// TwinCAT 3 PLC project RobustSolutionDemoProject
// ProgramVersion: 3.1.4026.24
// libraries:
//   [RobustSolution], * (BATW)
//   Tc2_MC2, * (Beckhoff Automation GmbH)
//   Tc2_Standard, * (Beckhoff Automation GmbH)
//   Tc2_System, * (Beckhoff Automation GmbH)
// project tree:
//   GVLs/ GVL_IO.TcGVL (not stored), GVL_Module.TcGVL (not stored), GVL_ShareMemory.TcGVL
//   / PlcTask.TcTTO
//   POUs/10_Chamber1/DUTs/Ctrl Status Interface/ ST_Chamber1_CtrlStatus.TcDUT (not stored), ST_Chamber1_ServiceCtrl.TcDUT, ST_Chamber1_ServiceParam.TcDUT, ST_Chamber1_ServiceStatus.TcDUT
//   POUs/10_Chamber1/DUTs/External IO/ ST_Chamber1_Signal_In.TcDUT, ST_Chamber1_Signal_Out.TcDUT
//   POUs/10_Chamber1/DUTs/ E_Chamber1ErrorCode.TcDUT, E_Chamber1ServiceId.TcDUT
//   POUs/10_Chamber1/DUTs/Service Param/Door/ ST_Chamber1DoorCloseParam.TcDUT, ST_Chamber1DoorOpenParam.TcDUT
//   POUs/10_Chamber1/DUTs/Service Param/Endpoint1PrepareWaferTransfer/ E_Ch1Ep1PrepareWaferTransferStep.TcDUT, ST_ChEp1PrepareWaferTransferParam.TcDUT
//   POUs/10_Chamber1/DUTs/Service Param/LiftAxis/ ST_Chamber1LiftPinAxisMoveAbsParam.TcDUT (not stored), ST_Chamber1LiftPinAxisMoveVelParam.TcDUT (not stored)
//   POUs/10_Chamber1/DUTs/Service Param/PreparePosition/ E_Chamber1PreparePositionStep.TcDUT, ST_Chamber1PreparePositionParam.TcDUT
//   POUs/10_Chamber1/DUTs/Service Param/SpinAxis/ ST_Chamber1SpinAxisJogParam.TcDUT (not stored), ST_Chamber1SpinAxisMoveAbsParam.TcDUT (not stored), ST_Chamber1SpinAxisMoveVelParam.TcDUT (not stored)
//   POUs/10_Chamber1/DUTs/Service Param/Vacuum/ ST_Chamber1VacuumOffParam.TcDUT, ST_Chamber1VacuumOnParam.TcDUT
//   POUs/10_Chamber1/ FB_Chamber1ModuleConfigurationAdapter.TcPOU, FB_Chamber1_Module.TcPOU
//   POUs/10_Chamber1/Services/Door/ FB_Chamber1Endpoint1DoorCloseService.TcPOU, FB_Chamber1Endpoint1DoorOpenService.TcPOU
//   POUs/10_Chamber1/Services/ FB_Chamber1PreparePositionService.TcPOU, FB_Chamber1Ep1PrepareWaferTransfer.TcPOU
//   POUs/10_Chamber1/Services/LiftAxis/ FB_Chamber1LiftPinAxisMoveAbsServices.TcPOU, FB_Chamber1LiftPinAxisMoveVelCCWServices.TcPOU, FB_Chamber1LiftPinAxisMoveVelCWServices.TcPOU
//   POUs/10_Chamber1/Services/SpinAxis/ FB_Chamber1SpinAxisJogCWServices.TcPOU, FB_Chamber1SpinAxisMoveAbsServices.TcPOU, FB_Chamber1SpinAxisMoveVelCWServices.TcPOU
//   POUs/10_Chamber1/Services/Vacuum/ FB_Chamber1VacuumOnService.TcPOU, FB_Chamber1VacuumOffService.TcPOU
//   POUs/ FB_ConfigRoot.TcPOU, MAIN.TcPOU (not stored)
// (motion and I/O tree: see PLC project robustsolutionframework)
// real-time tasks:
//   TASK UnitTest Task: cycle T#10ms, priority 21, ADS port 351
//   TASK DemoProject Task: cycle T#10ms, priority 22, ADS port 352
// variable links:
//   RobustSolutionDemoProject/RobustSolutionDemoProject Instance <-> NC-Task 1 SAF/Axes/Axis 1
//     PlcTask Inputs/GVL_IO.NC_Axis1._Axis.NcToPlc <-> Outputs/ToPlc
//     PlcTask Outputs/GVL_IO.NC_Axis1._Axis.PlcToNc <-> Inputs/FromPlc
//   RobustSolutionDemoProject/RobustSolutionDemoProject Instance <-> NC-Task 1 SAF/Axes/Axis 2
//     PlcTask Inputs/GVL_IO.NC_Axis2._Axis.NcToPlc <-> Outputs/ToPlc
//     PlcTask Outputs/GVL_IO.NC_Axis2._Axis.PlcToNc <-> Inputs/FromPlc

CONFIGURATION RobustSolutionDemoProject
    RESOURCE PLC ON TwinCAT3
        TASK PlcTask(INTERVAL := T#10ms, PRIORITY := 22);
        PROGRAM MAIN WITH PlcTask : MAIN;
    END_RESOURCE
END_CONFIGURATION

// ---- POUs/10_Chamber1/DUTs/Ctrl Status Interface/ST_Chamber1_ServiceCtrl.TcDUT
TYPE ST_Chamber1_ServiceCtrl :
STRUCT
	SpinAxisJogCW : ST_ServiceCtrl;
	SpinAxisMoveAbs : ST_ServiceCtrl;
	SpinAxisMoveVelCW	: ST_ServiceCtrl;
	LiftPinAxisMoveVelCW : ST_ServiceCtrl;
	LiftPinAxisMoveVelCCW : ST_ServiceCtrl;
	LiftPinAxisMoveAbs : ST_ServiceCtrl;
	
	DoorClose : ST_ServiceCtrl;
	DoorOpen : ST_ServiceCtrl;
	VacuumOn : ST_ServiceCtrl;
	VacuumOff : ST_ServiceCtrl;
	PreparePosition : ST_ServiceCtrl;
	Ep1PrepareWaferTransfer : ST_ServiceCtrl;
	SetMaterial : ST_ServiceCtrl;
END_STRUCT
END_TYPE

// ---- POUs/10_Chamber1/DUTs/Ctrl Status Interface/ST_Chamber1_ServiceParam.TcDUT
TYPE ST_Chamber1_ServiceParam :
STRUCT
	SpinAxisJogCW : ST_Chamber1SpinAxisJogParam;
	SpinAxisMoveAbs : ST_Chamber1SpinAxisMoveAbsParam;
	SpinAxisMoveVelCW : ST_Chamber1SpinAxisMoveVelParam;
	LiftPinAxisMoveVelCW : ST_Chamber1LiftPinAxisMoveVelParam;
	LiftPinAxisMoveVelCCW : ST_Chamber1LiftPinAxisMoveVelParam;
	LiftPinAxisMoveAbs : ST_Chamber1LiftPinAxisMoveAbsParam;
	DoorClose : ST_EmptyServiceParam;
	DoorOpen : ST_EmptyServiceParam;
	VacuumOn : ST_EmptyServiceParam;
	VacuumOff : ST_EmptyServiceParam;
	PreparePosition : ST_Chamber1PreparePositionParam;
	Ep1PrepareWaferTransfer : ST_EmptyServiceParam;
	SetMaterialParam : ST_MaterialParam;
END_STRUCT
END_TYPE

// ---- POUs/10_Chamber1/DUTs/Ctrl Status Interface/ST_Chamber1_ServiceStatus.TcDUT
TYPE ST_Chamber1_ServiceStatus :
STRUCT
	SpinAxisJogCW : ST_ServiceStatus;
	SpinAxisMoveAbs : ST_ServiceStatus;
	SpinAxisMoveVelCW : ST_ServiceStatus;
	LiftPinAxisMoveVelCW : ST_ServiceStatus;
	LiftPinAxisMoveVelCCW : ST_ServiceStatus;
	LiftPinAxisMoveAbs : ST_ServiceStatus;
	DoorClose : ST_ServiceStatus;
	DoorOpen : ST_ServiceStatus;
	VacuumOn : ST_ServiceStatus;
	VacuumOff : ST_ServiceStatus;
	PreparePosition : ST_ServiceStatus;
	Ep1PrepareWaferTransfer : ST_ServiceStatus;
	SetMaterial : ST_ServiceStatus;
END_STRUCT
END_TYPE

// ---- POUs/10_Chamber1/DUTs/External IO/ST_Chamber1_Signal_In.TcDUT
TYPE ST_Chamber1_Signal_In :
STRUCT
	bDoorClosed : BOOL;
	bVacuumOn : BOOL;
	rTemperature : REAL;
	bRobotInChamber : BOOL;

	bDIs : ARRAY[1..16] OF BOOL;
	rAIs : ARRAY[1..16] OF REAL;
END_STRUCT
END_TYPE

// ---- POUs/10_Chamber1/DUTs/External IO/ST_Chamber1_Signal_Out.TcDUT
TYPE ST_Chamber1_Signal_Out :
STRUCT
	bDoorClosed : BOOL;
	bVaccumOn : BOOL;

	bDOs : ARRAY[1..16] OF BOOL;
	rAOs : ARRAY[1..16] OF REAL;
END_STRUCT
END_TYPE

// ---- POUs/10_Chamber1/DUTs/E_Chamber1ErrorCode.TcDUT
{attribute 'qualified_only'}
{attribute 'to_string'}
TYPE E_Chamber1ErrorCode :
(
	None := 0,
	Axis_Not_Servo_On_During_Starting := 1,
	Axis_Is_Busy_During_Starting := 2,
	Invalid_Param := 3,
	Axis_Command_Error_During_Execute := 4,
	Error_While_Stop_Axis := 5,
	// The BaseUnit was already owned by another Service.
	Resource_Acquire_Failed_During_Starting := 6,
	// The asynchronous Reset used while aborting failed.
	Error_While_Reset_Axis := 7,
	Close_Door_While_Robot_In_Chamber := 8
)UDINT;
END_TYPE

// ---- POUs/10_Chamber1/DUTs/E_Chamber1ServiceId.TcDUT
{attribute 'qualified_only'}
{attribute 'to_string'}
TYPE E_Chamber1ServiceId :
(
	// Each value identifies one Service instance within the Chamber1 Module.
	None := 0,
	SpinAxisJogCW := 1,
	SpinAxisMoveAbs := 2,
	SpinAxisMoveVelCW := 3,
	LiftPinAxisMoveVelCW := 4,
	LiftPinAxisMoveVelCCW := 5,
	LiftPinAxisMoveAbs := 6,
	Endpoint1PrepareSendWafer := 8,
	DoorOpen := 9,
	DoorClose := 10,
	VacuumOn := 11,
	VacuumOff := 12,
	PreparePosition := 13,
	SetMaterial := 14
) UDINT;
END_TYPE

// ---- POUs/10_Chamber1/DUTs/Service Param/Door/ST_Chamber1DoorCloseParam.TcDUT
TYPE ST_Chamber1DoorCloseParam :
STRUCT
END_STRUCT
END_TYPE

// ---- POUs/10_Chamber1/DUTs/Service Param/Door/ST_Chamber1DoorOpenParam.TcDUT
TYPE ST_Chamber1DoorOpenParam :
STRUCT
END_STRUCT
END_TYPE

// ---- POUs/10_Chamber1/DUTs/Service Param/Endpoint1PrepareWaferTransfer/E_Ch1Ep1PrepareWaferTransferStep.TcDUT
{attribute 'qualified_only'}
{attribute 'strict'}
{attribute 'to_string'}
TYPE E_Ch1Ep1PrepareWaferTransferStep :
(
	None := 0,
	MoveLiftPinAxis := 1,
	VacuumOff := 2,
	Finish := 3
) UDINT;
END_TYPE

// ---- POUs/10_Chamber1/DUTs/Service Param/Endpoint1PrepareWaferTransfer/ST_ChEp1PrepareWaferTransferParam.TcDUT
TYPE ST_ChEp1PrepareWaferTransferParam :
STRUCT
END_STRUCT
END_TYPE

// ---- POUs/10_Chamber1/DUTs/Service Param/PreparePosition/E_Chamber1PreparePositionStep.TcDUT
{attribute 'qualified_only'}
{attribute 'strict'}
{attribute 'to_string'}
TYPE E_Chamber1PreparePositionStep :
(
	None := 0,
	LiftReady := 1,
	SpinAlign := 2,
	ResetLift := 3,
	LiftWork := 4,
	Finish := 5
) UDINT;
END_TYPE

// ---- POUs/10_Chamber1/DUTs/Service Param/PreparePosition/ST_Chamber1PreparePositionParam.TcDUT
TYPE ST_Chamber1PreparePositionParam :
STRUCT
	LiftReadyPosition : LREAL;
	LiftReadyVelocity : LREAL;
	LiftReadyAcceleration : LREAL;
	LiftReadyDeceleration : LREAL;
	SpinAlignPosition : LREAL;
	SpinAlignVelocity : LREAL;
	SpinAlignAcceleration : LREAL;
	SpinAlignDeceleration : LREAL;
	LiftWorkPosition : LREAL;
	LiftWorkVelocity : LREAL;
	LiftWorkAcceleration : LREAL;
	LiftWorkDeceleration : LREAL;
END_STRUCT
END_TYPE

// ---- POUs/10_Chamber1/DUTs/Service Param/Vacuum/ST_Chamber1VacuumOffParam.TcDUT
TYPE ST_Chamber1VacuumOffParam :
STRUCT
END_STRUCT
END_TYPE

// ---- POUs/10_Chamber1/DUTs/Service Param/Vacuum/ST_Chamber1VacuumOnParam.TcDUT
TYPE ST_Chamber1VacuumOnParam :
STRUCT
END_STRUCT
END_TYPE

// ---- GVLs/GVL_ShareMemory.TcGVL
{attribute 'qualified_only'}
VAR_GLOBAL
	bChamber1_Endpoint1_DoorClosed : BOOL;
	bChamber1_VacuumOn : BOOL;
	
	bRobotIsInChamber1 : BOOL;
END_VAR

// ---- POUs/10_Chamber1/FB_Chamber1ModuleConfigurationAdapter.TcPOU
FUNCTION_BLOCK FB_Chamber1ModuleConfigurationAdapter IMPLEMENTS I_ModuleConfigurationAdapter

METHOD PUBLIC M_ApplyRuntimeConfig : BOOL
VAR_INPUT
	Slot : UINT;
END_VAR
VAR_IN_OUT CONSTANT
	RuntimeConfig : ST_ModuleRuntimeConfig;
END_VAR
VAR_OUTPUT
	ErrorMessage : STRING(255);
END_VAR
M_ApplyRuntimeConfig := FALSE;
ErrorMessage := '';
IF NOT M_IsSlotSupported(Slot := Slot) THEN
	ErrorMessage := 'Chamber1 slot is outside the supported range.';
	RETURN;
END_IF
IF RuntimeConfig.ModuleType <> 'Chamber1' THEN
	ErrorMessage := 'Runtime configuration type is incompatible with the Chamber1 adapter.';
	RETURN;
END_IF
GVL_Module.Chamber1_Runtime[Slot] := RuntimeConfig;
M_ApplyRuntimeConfig := TRUE;
END_METHOD

METHOD PUBLIC M_ClearAllSlots : BOOL
VAR_OUTPUT
	ErrorMessage : STRING(255);
END_VAR
VAR
	nSlot : UINT;
END_VAR
M_ClearAllSlots := FALSE;
ErrorMessage := '';
FOR nSlot := 1 TO Param_Config.MaxModulePerType DO
	GVL_Module.Chamber1_SpinAxis[nSlot] := 0;
	GVL_Module.Chamber1_LiftPinAxis[nSlot] := 0;
	MEMSET(ADR(GVL_Module.Chamber1_Runtime[nSlot]), 0, SIZEOF(GVL_Module.Chamber1_Runtime[nSlot]));
END_FOR
M_ClearAllSlots := TRUE;
END_METHOD

METHOD PUBLIC M_IsSlotSupported : BOOL
VAR_INPUT
	Slot : UINT;
END_VAR
M_IsSlotSupported := (Slot >= 1) AND (Slot <= Param_Config.MaxModulePerType);
END_METHOD

METHOD PUBLIC M_PrepareInstance : BOOL
VAR_INPUT
	Slot : UINT;
	ReferenceBindings : I_ModuleReferenceBindings;
END_VAR
VAR_IN_OUT
	ModuleConfig : ST_ModuleFileConfig;
	LinkVariableManager : FB_LinkVariableManager;
END_VAR
VAR_OUTPUT
	ModuleSymbol : STRING(255);
	ErrorMessage : STRING(255);
END_VAR
VAR
	bDeclared : BOOL;
	BaseUnit : I_BaseUnit;
	SpinAxis : I_Axis_BaseUnit;
	LiftPinAxis : I_Axis_BaseUnit;
	sReferenceError : STRING(255);
	sPortName : STRING(80);
	nIndex : DINT;
END_VAR
M_PrepareInstance := FALSE;
ModuleSymbol := '';
ErrorMessage := '';
IF NOT M_IsSlotSupported(Slot := Slot) THEN
	ErrorMessage := 'Chamber1 slot is outside the supported range.';
	RETURN;
END_IF

// Register module hardware I/O as link node
bDeclared := LinkVariableManager.M_BeginModuleRegistration(
	Address := ADR(GVL_Module.Chamber1[Slot]),
	Size := SIZEOF(GVL_Module.Chamber1[Slot]),
	ModuleConfig := ModuleConfig);

bDeclared := LinkVariableManager.M_RegisterModuleNode(
	Variable := GVL_Module.Chamber1[Slot].HwInput.bDoorClosed,
	Access := E_VariableAccess.ReadWrite);
bDeclared := LinkVariableManager.M_RegisterModuleNode(
	Variable := GVL_Module.Chamber1[Slot].HwInput.bVacuumOn,
	Access := E_VariableAccess.ReadWrite);
bDeclared := LinkVariableManager.M_RegisterModuleNode(
	Variable := GVL_Module.Chamber1[Slot].HwInput.bRobotInChamber,
	Access := E_VariableAccess.ReadWrite);
bDeclared := LinkVariableManager.M_RegisterModuleNode(
	Variable := GVL_Module.Chamber1[Slot].HwInput.rTemperature,
	Access := E_VariableAccess.ReadWrite);

FOR nIndex := LOWER_BOUND(GVL_Module.Chamber1[Slot].HwInput.bDIs, 1)
	TO UPPER_BOUND(GVL_Module.Chamber1[Slot].HwInput.bDIs, 1) DO
	bDeclared := LinkVariableManager.M_RegisterModuleNode(
		Variable := GVL_Module.Chamber1[Slot].HwInput.bDIs[nIndex],
		Access := E_VariableAccess.ReadWrite);
END_FOR
FOR nIndex := LOWER_BOUND(GVL_Module.Chamber1[Slot].HwInput.rAIs, 1)
	TO UPPER_BOUND(GVL_Module.Chamber1[Slot].HwInput.rAIs, 1) DO
	bDeclared := LinkVariableManager.M_RegisterModuleNode(
		Variable := GVL_Module.Chamber1[Slot].HwInput.rAIs[nIndex],
		Access := E_VariableAccess.ReadWrite);
END_FOR

bDeclared := LinkVariableManager.M_RegisterModuleNode(
	Variable := GVL_Module.Chamber1[Slot].HwOutput.bVaccumOn,
	Access := E_VariableAccess.ReadOnly);
bDeclared := LinkVariableManager.M_RegisterModuleNode(
	Variable := GVL_Module.Chamber1[Slot].HwOutput.bDoorClosed,
	Access := E_VariableAccess.ReadOnly);
	
FOR nIndex := LOWER_BOUND(GVL_Module.Chamber1[Slot].HwOutput.bDOs, 1)
	TO UPPER_BOUND(GVL_Module.Chamber1[Slot].HwOutput.bDOs, 1) DO
	bDeclared := LinkVariableManager.M_RegisterModuleNode(
		Variable := GVL_Module.Chamber1[Slot].HwOutput.bDOs[nIndex],
		Access := E_VariableAccess.ReadOnly);
END_FOR
FOR nIndex := LOWER_BOUND(GVL_Module.Chamber1[Slot].HwOutput.rAOs, 1)
	TO UPPER_BOUND(GVL_Module.Chamber1[Slot].HwOutput.rAOs, 1) DO
	bDeclared := LinkVariableManager.M_RegisterModuleNode(
		Variable := GVL_Module.Chamber1[Slot].HwOutput.rAOs[nIndex],
		Access := E_VariableAccess.ReadOnly);
END_FOR

IF NOT LinkVariableManager.M_EndModuleRegistration(ModuleSymbol => ModuleSymbol) THEN
	ErrorMessage := LinkVariableManager.ErrorMessage;
	RETURN;
END_IF

// Bind base-unit instance to module-base-unit interface
IF ReferenceBindings = 0 THEN
	ErrorMessage := 'Chamber1 requires a Module reference binding context.';
	RETURN;
END_IF

IF NOT ReferenceBindings.M_SetModuleScope(
	ModuleSymbol := ModuleSymbol,
	ErrorMessage => sReferenceError) THEN
	ErrorMessage := sReferenceError;
	RETURN;
END_IF

BaseUnit := ReferenceBindings.M_TakeRequired(
	Port := GVL_Module.Chamber1[Slot].SpinAxis_BaseUnit,
	PortName => sPortName,
	ErrorMessage => sReferenceError);
IF BaseUnit = 0 THEN
	ErrorMessage := sReferenceError;
	RETURN;
END_IF
SpinAxis := 0;
IF NOT __QUERYINTERFACE(BaseUnit, SpinAxis) THEN
	ErrorMessage := CONCAT(sPortName, ' requires I_Axis_BaseUnit.');
	RETURN;
END_IF

BaseUnit := ReferenceBindings.M_TakeRequired(
	Port := GVL_Module.Chamber1[Slot].LiftPinAxis_BaseUnit,
	PortName => sPortName,
	ErrorMessage => sReferenceError);
IF BaseUnit = 0 THEN
	ErrorMessage := sReferenceError;
	RETURN;
END_IF
LiftPinAxis := 0;
IF NOT __QUERYINTERFACE(BaseUnit, LiftPinAxis) THEN
	ErrorMessage := CONCAT(sPortName, ' requires I_Axis_BaseUnit.');
	RETURN;
END_IF

// Commit typed references only after the complete Chamber1 reference contract is valid.
GVL_Module.Chamber1_SpinAxis[Slot] := SpinAxis;
GVL_Module.Chamber1_LiftPinAxis[Slot] := LiftPinAxis;
M_PrepareInstance := TRUE;
END_METHOD

END_FUNCTION_BLOCK

// ---- POUs/10_Chamber1/FB_Chamber1_Module.TcPOU
FUNCTION_BLOCK FB_Chamber1_Module EXTENDS FB_ModuleBase
VAR_INPUT	
	HwInput : ST_Chamber1_Signal_In;

	ServiceCtrl : REFERENCE TO ST_Chamber1_ServiceCtrl;
	ServiceParam : REFERENCE TO ST_Chamber1_ServiceParam;

	// Base unit used in Chamber1 chamber
	SpinAxis_BaseUnit : I_Axis_BaseUnit;
	LiftPinAxis_BaseUnit : I_Axis_BaseUnit;
END_VAR

VAR_OUTPUT
	HwOutput : ST_Chamber1_Signal_Out;
	ServiceStatus : ST_Chamber1_ServiceStatus;
END_VAR

VAR
	_EffectiveServiceCtrl : ST_Chamber1_ServiceCtrl;
	_EffectiveServiceParam : ST_Chamber1_ServiceParam;
	_ServiceStatusStore : ST_Chamber1_ServiceStatus;

	_SpinAxisJogCWService : FB_Chamber1SpinAxisJogCWServices;
	_SpinAxisMoveAbsService : FB_Chamber1SpinAxisMoveAbsServices;
	_SpinAxisMoveVelCWService : FB_Chamber1SpinAxisMoveVelCWServices;
	_LiftPinAxisMoveVelCWService : FB_Chamber1LiftPinAxisMoveVelCWServices;
	_LiftPinAxisMoveVelCCWService : FB_Chamber1LiftPinAxisMoveVelCCWServices;
	_LiftPinAxisMoveAbsService : FB_Chamber1LiftPinAxisMoveAbsServices;
	_Endpoint1DoorOpenService : FB_Chamber1Endpoint1DoorOpenService;
	_Endpoint1DoorCloseService : FB_Chamber1Endpoint1DoorCloseService;
	_VacuumOffService : FB_Chamber1VacuumOffService;
	_VacuumOnService : FB_Chamber1VacuumOnService;
	_Ep1PrepareWaferTransferService : FB_Chamber1Ep1PrepareWaferTransfer;
	_PreparePositionService : FB_Chamber1PreparePositionService;
	_SetMaterialService : FB_SetMaterialService;
	
	_bEndpoint1_SendReady : BOOL;
	_bEndpoint1_SendPrepared : BOOL;
	_bEndpoint1_ReceiveReady : BOOL;
	_bEndpoint1_ReceivePrepared : BOOL;
END_VAR

// An unbound Axis interface is a composition error. Keep the Module inert.
IF (SpinAxis_BaseUnit = 0) OR (LiftPinAxis_BaseUnit = 0) THEN
	RETURN;
END_IF

// Config wafer transfer endpoint
ModuleStatus.WaferStatusList[1].EndpointId := 1;
ModuleStatus.WaferStatusList[1].EndpointName := 'Hello World';

// Update endpoint status (for SVID display)
_bEndpoint1_SendReady := _ServiceCoordinator.AllIdle AND
						 ModuleStatus.WaferStatusList[1].MaterialContext.Id <> '';
						 
_bEndpoint1_SendPrepared := _bEndpoint1_SendReady AND
							HwInput.bVacuumOn = FALSE AND
							LiftPinAxis_BaseUnit.AxisActualPosition = 70.0;

_bEndpoint1_ReceiveReady := _ServiceCoordinator.AllIdle AND
						 ModuleStatus.WaferStatusList[1].MaterialContext.Id = '';
						 
_bEndpoint1_ReceivePrepared := _bEndpoint1_ReceiveReady AND
							HwInput.bVacuumOn = FALSE AND
							LiftPinAxis_BaseUnit.AxisActualPosition = 70.0;

M_UpdateModule();

// Update status
ServiceStatus := _ServiceStatusStore;

METHOD PROTECTED H_RegisterServices
// Register services
M_RegisterService(
	ServiceId := E_Chamber1ServiceId.SpinAxisJogCW,
	AllowCompositeCall := TRUE,
	UpperCtrl := ServiceCtrl.SpinAxisJogCW,
	EffectiveCtrl := _EffectiveServiceCtrl.SpinAxisJogCW,
	UpperParam := ServiceParam.SpinAxisJogCW,
	EffectiveParam := _EffectiveServiceParam.SpinAxisJogCW,
	Status := _ServiceStatusStore.SpinAxisJogCW);
M_RegisterService(
	ServiceId := E_Chamber1ServiceId.SpinAxisMoveAbs,
	AllowCompositeCall := TRUE,
	UpperCtrl := ServiceCtrl.SpinAxisMoveAbs,
	EffectiveCtrl := _EffectiveServiceCtrl.SpinAxisMoveAbs,
	UpperParam := ServiceParam.SpinAxisMoveAbs,
	EffectiveParam := _EffectiveServiceParam.SpinAxisMoveAbs,
	Status := _ServiceStatusStore.SpinAxisMoveAbs);
M_RegisterService(
	ServiceId := E_Chamber1ServiceId.SpinAxisMoveVelCW,
	AllowCompositeCall := TRUE,
	UpperCtrl := ServiceCtrl.SpinAxisMoveVelCW,
	EffectiveCtrl := _EffectiveServiceCtrl.SpinAxisMoveVelCW,
	UpperParam := ServiceParam.SpinAxisMoveVelCW,
	EffectiveParam := _EffectiveServiceParam.SpinAxisMoveVelCW,
	Status := _ServiceStatusStore.SpinAxisMoveVelCW);
M_RegisterService(
	ServiceId := E_Chamber1ServiceId.LiftPinAxisMoveVelCW,
	AllowCompositeCall := TRUE,
	UpperCtrl := ServiceCtrl.LiftPinAxisMoveVelCW,
	EffectiveCtrl := _EffectiveServiceCtrl.LiftPinAxisMoveVelCW,
	UpperParam := ServiceParam.LiftPinAxisMoveVelCW,
	EffectiveParam := _EffectiveServiceParam.LiftPinAxisMoveVelCW,
	Status := _ServiceStatusStore.LiftPinAxisMoveVelCW);
M_RegisterService(
	ServiceId := E_Chamber1ServiceId.LiftPinAxisMoveVelCCW,
	AllowCompositeCall := TRUE,
	UpperCtrl := ServiceCtrl.LiftPinAxisMoveVelCCW,
	EffectiveCtrl := _EffectiveServiceCtrl.LiftPinAxisMoveVelCCW,
	UpperParam := ServiceParam.LiftPinAxisMoveVelCCW,
	EffectiveParam := _EffectiveServiceParam.LiftPinAxisMoveVelCCW,
	Status := _ServiceStatusStore.LiftPinAxisMoveVelCCW);
M_RegisterService(
	ServiceId := E_Chamber1ServiceId.LiftPinAxisMoveAbs,
	AllowCompositeCall := TRUE,
	UpperCtrl := ServiceCtrl.LiftPinAxisMoveAbs,
	EffectiveCtrl := _EffectiveServiceCtrl.LiftPinAxisMoveAbs,
	UpperParam := ServiceParam.LiftPinAxisMoveAbs,
	EffectiveParam := _EffectiveServiceParam.LiftPinAxisMoveAbs,
	Status := _ServiceStatusStore.LiftPinAxisMoveAbs);
M_RegisterService(
	ServiceId := E_Chamber1ServiceId.DoorClose,
	AllowCompositeCall := TRUE,
	UpperCtrl := ServiceCtrl.DoorClose,
	EffectiveCtrl := _EffectiveServiceCtrl.DoorClose,
	UpperParam := ServiceParam.DoorClose,
	EffectiveParam := _EffectiveServiceParam.DoorClose,
	Status := _ServiceStatusStore.DoorClose);
M_RegisterService(
	ServiceId := E_Chamber1ServiceId.DoorOpen,
	AllowCompositeCall := TRUE,
	UpperCtrl := ServiceCtrl.DoorOpen,
	EffectiveCtrl := _EffectiveServiceCtrl.DoorOpen,
	UpperParam := ServiceParam.DoorOpen,
	EffectiveParam := _EffectiveServiceParam.DoorOpen,
	Status := _ServiceStatusStore.DoorOpen);
M_RegisterService(
	ServiceId := E_Chamber1ServiceId.VacuumOff,
	AllowCompositeCall := TRUE,
	UpperCtrl := ServiceCtrl.VacuumOff,
	EffectiveCtrl := _EffectiveServiceCtrl.VacuumOff,
	UpperParam := ServiceParam.VacuumOff,
	EffectiveParam := _EffectiveServiceParam.VacuumOff,
	Status := _ServiceStatusStore.VacuumOff);
M_RegisterService(
	ServiceId := E_Chamber1ServiceId.VacuumOn,
	AllowCompositeCall := TRUE,
	UpperCtrl := ServiceCtrl.VacuumOn,
	EffectiveCtrl := _EffectiveServiceCtrl.VacuumOn,
	UpperParam := ServiceParam.VacuumOn,
	EffectiveParam := _EffectiveServiceParam.VacuumOn,
	Status := _ServiceStatusStore.VacuumOn);
M_RegisterService(
	ServiceId := E_Chamber1ServiceId.PreparePosition,
	AllowCompositeCall := FALSE,
	UpperCtrl := ServiceCtrl.PreparePosition,
	EffectiveCtrl := _EffectiveServiceCtrl.PreparePosition,
	UpperParam := ServiceParam.PreparePosition,
	EffectiveParam := _EffectiveServiceParam.PreparePosition,
	Status := _ServiceStatusStore.PreparePosition);
M_RegisterService(
	ServiceId := E_Chamber1ServiceId.Endpoint1PrepareSendWafer,
	AllowCompositeCall := FALSE,
	UpperCtrl := ServiceCtrl.Ep1PrepareWaferTransfer,
	EffectiveCtrl := _EffectiveServiceCtrl.Ep1PrepareWaferTransfer,
	UpperParam := ServiceParam.Ep1PrepareWaferTransfer,
	EffectiveParam := _EffectiveServiceParam.Ep1PrepareWaferTransfer,
	Status := _ServiceStatusStore.Ep1PrepareWaferTransfer);
M_RegisterService(
	ServiceId := E_Chamber1ServiceId.SetMaterial,
	AllowCompositeCall := TRUE,
	UpperCtrl := ServiceCtrl.SetMaterial,
	EffectiveCtrl := _EffectiveServiceCtrl.SetMaterial,
	UpperParam := ServiceParam.SetMaterialParam,
	EffectiveParam := _EffectiveServiceParam.SetMaterialParam,
	Status := _ServiceStatusStore.SetMaterial);

// Register dependency of composite service
_PreparePositionService.M_RegisterDefinition(
	CompositeServiceId := E_Chamber1ServiceId.PreparePosition,
	Coordinator := _ServiceCoordinator);
_Ep1PrepareWaferTransferService.M_RegisterDefinition(
	CompositeServiceId := E_Chamber1ServiceId.Endpoint1PrepareSendWafer,
	Coordinator := _ServiceCoordinator);
END_METHOD

METHOD PROTECTED H_UpdateBaseUnit
VAR_INPUT
END_VAR
SpinAxis_BaseUnit.M_CyclicUpdate();
LiftPinAxis_BaseUnit.M_CyclicUpdate();
END_METHOD

METHOD PROTECTED H_UpdateService
VAR_INPUT
END_VAR
_SpinAxisJogCWService(
	Ctrl:= _EffectiveServiceCtrl.SpinAxisJogCW,
	Param:= _EffectiveServiceParam.SpinAxisJogCW,
	Context:= _ServiceContext,
	Axis_BaseUnit:= SpinAxis_BaseUnit,
	// Owner IDs are assigned by the Module so each Service instance is unique.
	ServiceId:= E_Chamber1ServiceId.SpinAxisJogCW,
	Status=> _ServiceStatusStore.SpinAxisJogCW);

_SpinAxisMoveAbsService(
	Ctrl:= _EffectiveServiceCtrl.SpinAxisMoveAbs,
	Param:= _EffectiveServiceParam.SpinAxisMoveAbs,
	Context:= _ServiceContext,
	Axis_BaseUnit:= SpinAxis_BaseUnit,
	ServiceId:= E_Chamber1ServiceId.SpinAxisMoveAbs,
	Status=> _ServiceStatusStore.SpinAxisMoveAbs);

_SpinAxisMoveVelCWService(
	Ctrl:= _EffectiveServiceCtrl.SpinAxisMoveVelCW,
	Param:= _EffectiveServiceParam.SpinAxisMoveVelCW,
	Context:= _ServiceContext,
	Axis_BaseUnit:= SpinAxis_BaseUnit,
	ServiceId:= E_Chamber1ServiceId.SpinAxisMoveVelCW,
	Status=> _ServiceStatusStore.SpinAxisMoveVelCW);

_LiftPinAxisMoveVelCWService(
	Ctrl:= _EffectiveServiceCtrl.LiftPinAxisMoveVelCW,
	Param:= _EffectiveServiceParam.LiftPinAxisMoveVelCW,
	Context:= _ServiceContext,
	Axis_BaseUnit:= LiftPinAxis_BaseUnit,
	ServiceId:= E_Chamber1ServiceId.LiftPinAxisMoveVelCW,
	Status=> _ServiceStatusStore.LiftPinAxisMoveVelCW);

_LiftPinAxisMoveVelCCWService(
	Ctrl:= _EffectiveServiceCtrl.LiftPinAxisMoveVelCCW,
	Param:= _EffectiveServiceParam.LiftPinAxisMoveVelCCW,
	Context:= _ServiceContext,
	Axis_BaseUnit:= LiftPinAxis_BaseUnit,
	ServiceId:= E_Chamber1ServiceId.LiftPinAxisMoveVelCCW,
	Status=> _ServiceStatusStore.LiftPinAxisMoveVelCCW);

_LiftPinAxisMoveAbsService(
	Ctrl:= _EffectiveServiceCtrl.LiftPinAxisMoveAbs,
	Param:= _EffectiveServiceParam.LiftPinAxisMoveAbs,
	Context:= _ServiceContext,
	Axis_BaseUnit:= LiftPinAxis_BaseUnit,
	ServiceId:= E_Chamber1ServiceId.LiftPinAxisMoveAbs,
	Status=> _ServiceStatusStore.LiftPinAxisMoveAbs);
	
_Endpoint1DoorOpenService(
	Ctrl:=  _EffectiveServiceCtrl.DoorOpen, 
	Context:= _ServiceContext, 
	ServiceId:= E_Chamber1ServiceId.DoorOpen, 
	Status=> _ServiceStatusStore.DoorOpen, 
	IsDoorClose:= HwInput.bDoorClosed, 
	DoorCloseCtrl:= HwOutput.bDoorClosed);

_Endpoint1DoorCloseService(
	Ctrl:=  _EffectiveServiceCtrl.DoorClose, 
	Context:= _ServiceContext, 
	ServiceId:= E_Chamber1ServiceId.DoorClose, 
	Status=> _ServiceStatusStore.DoorClose, 
	IsDoorClose:= HwInput.bDoorClosed,
	IsRobotInChamber:= HwInput.bRobotInChamber,
	DoorCloseCtrl:= HwOutput.bDoorClosed);
	
_VacuumOnService(
	Ctrl:= _EffectiveServiceCtrl.VacuumOn, 
	Context:= _ServiceContext, 
	ServiceId:= E_Chamber1ServiceId.VacuumOn, 
	Status=> _ServiceStatusStore.VacuumOn, 
	IsVacuumOn:= HwInput.bVacuumOn, 
	VacuumOnCtrl:= HwOutput.bVaccumOn);
	
_VacuumOffService(
	Ctrl:= _EffectiveServiceCtrl.VacuumOff, 
	Context:= _ServiceContext, 
	ServiceId:= E_Chamber1ServiceId.VacuumOff, 
	Status=> _ServiceStatusStore.VacuumOff, 
	IsVacuumOn:= HwInput.bVacuumOn, 
	VacuumOnCtrl:= HwOutput.bVaccumOn);

_SetMaterialService(
	Ctrl:= _EffectiveServiceCtrl.SetMaterial,
	Context:= _ServiceContext,
	ServiceId:= E_Chamber1ServiceId.SetMaterial,
	Status=> _ServiceStatusStore.SetMaterial,
	Param:= _EffectiveServiceParam.SetMaterialParam,
	WaferStatusList:= ModuleStatus.WaferStatusList);

_PreparePositionService(
	Ctrl := _EffectiveServiceCtrl.PreparePosition,
	Param:= _EffectiveServiceParam.PreparePosition,
	Context := _ServiceContext,
	ServiceId := E_Chamber1ServiceId.PreparePosition,
	Status => _ServiceStatusStore.PreparePosition);

_Ep1PrepareWaferTransferService(
	Ctrl:= _EffectiveServiceCtrl.Ep1PrepareWaferTransfer, 
	Context:= _ServiceContext, 
	ServiceId:= E_Chamber1ServiceId.Endpoint1PrepareSendWafer, 
	Status=> _ServiceStatusStore.Ep1PrepareWaferTransfer);
END_METHOD

METHOD PROTECTED H_UpdateVariable
M_AddVariable(Id:= 10, Name:= 'Endpoint1_SendReady', DataType:= E_DescriptorType.Boolean, Unit:= '', Value:= TO_STRING(_bEndpoint1_SendReady));
M_AddVariable(Id:= 11, Name:= 'Endpoint1_SendPrepared', DataType:= E_DescriptorType.Boolean, Unit:= '', Value:= TO_STRING(_bEndpoint1_SendPrepared));
M_AddVariable(Id:= 12, Name:= 'Endpoint1_ReceiveReady', DataType:= E_DescriptorType.Boolean, Unit:= '', Value:= TO_STRING(_bEndpoint1_ReceiveReady));
M_AddVariable(Id:= 13, Name:= 'Endpoint1_ReceivePrepared', DataType:= E_DescriptorType.Boolean, Unit:= '', Value:= TO_STRING(_bEndpoint1_ReceivePrepared));
END_METHOD

END_FUNCTION_BLOCK

// ---- POUs/10_Chamber1/Services/SpinAxis/FB_Chamber1SpinAxisJogCWServices.TcPOU
FUNCTION_BLOCK FB_Chamber1SpinAxisJogCWServices EXTENDS FB_ServiceBase
VAR_INPUT
	Param : ST_Chamber1SpinAxisJogParam;
	Axis_BaseUnit : I_Axis_BaseUnit;
END_VAR

M_UpdateService(CompletionBehavior := E_ServiceCompletionBehavior.ExecuteUntilExternalStop);

METHOD PROTECTED H_OnAborted
VAR_INPUT
	bFirstScan	: BOOL;
END_VAR
// Release defensively in case an unexpected transition skipped cleanup.
Axis_BaseUnit.M_ReleaseResource(OwnerId := ServiceId);
END_METHOD

METHOD PROTECTED H_OnAborting : E_PackMLHookResult
VAR_INPUT
	bFirstScan	: BOOL;
END_VAR
H_OnAborting := E_PackMLHookResult.Done;

// A Service that never acquired the Resource must not affect its Owner.
IF NOT Axis_BaseUnit.M_IsResourceOwner(OwnerId := ServiceId) THEN
	RETURN;
END_IF

Axis_BaseUnit.M_Jog(
	OwnerId:= ServiceId,
	JogForward:= FALSE, 
	JogBackwards:= FALSE, 
	Mode:= E_JogMode.MC_JOGMODE_CONTINOUS,
	Position:= Param.Position,
	Velocity:= Param.Velocity,
	Acceleration:= Param.Acceleration,
	Deceleration:= Param.Deceleration);

// Jog has no asynchronous abort phase once both direction commands are false.
Axis_BaseUnit.M_ReleaseResource(OwnerId := ServiceId);
END_METHOD

METHOD PROTECTED H_OnClearing : E_PackMLHookResult
VAR_INPUT
	bFirstScan	: BOOL;
END_VAR

VAR
	bServoOn : BOOL;
	bError : BOOL;
	nErrorId : UDINT;
END_VAR
M_ClearAllError();
H_OnClearing := E_PackMLHookResult.Done;
END_METHOD

METHOD PROTECTED H_OnComplete
VAR_INPUT
	bFirstScan	: BOOL;
END_VAR
// Completing normally releases first; this is an idempotent safety net.
Axis_BaseUnit.M_ReleaseResource(OwnerId := ServiceId);
END_METHOD

METHOD PROTECTED H_OnCompleting : E_PackMLHookResult
VAR_INPUT
	bFirstScan	: BOOL;
END_VAR
Axis_BaseUnit.M_Jog(
	OwnerId:= ServiceId,
	JogForward:= FALSE, 
	JogBackwards:= FALSE, 
	Mode:= E_JogMode.MC_JOGMODE_CONTINOUS,
	Position:= Param.Position,
	Velocity:= Param.Velocity,
	Acceleration:= Param.Acceleration,
	Deceleration:= Param.Deceleration);

// Release only after the active Jog request has been withdrawn.
Axis_BaseUnit.M_ReleaseResource(OwnerId := ServiceId);
H_OnCompleting := E_PackMLHookResult.Done;
END_METHOD

METHOD PROTECTED H_OnExecute : E_PackMLHookResult
VAR_INPUT
	bFirstScan	: BOOL;
END_VAR

VAR
	bError : BOOL;
	nErrorId : UDINT;
END_VAR
H_OnExecute := E_PackMLHookResult.Busy;

Axis_BaseUnit.M_Jog(
	OwnerId:= ServiceId,
	JogForward:= TRUE,
	JogBackwards:= FALSE,
	Mode:= E_JogMode.MC_JOGMODE_CONTINOUS,
	Position:= Param.Position,
	Velocity:= Param.Velocity,
	Acceleration:= Param.Acceleration,
	Deceleration:= Param.Deceleration,
	Done=> , Error=> bError, ErrorId=> nErrorId);


IF bError THEN
	M_AddError(
		MainErrorId := E_Chamber1ErrorCode.Axis_Command_Error_During_Execute,
		SourceErrorId := nErrorId,
		Message := 'Jog failed during Execute.');
	RequestCommand(E_PackMLCommand.Abort);
END_IF
END_METHOD

METHOD PROTECTED H_OnIdle
VAR_INPUT
	bFirstScan	: BOOL;
END_VAR
// Idle Services must not retain a Resource from an earlier operation.
Axis_BaseUnit.M_ReleaseResource(OwnerId := ServiceId);
END_METHOD

METHOD PROTECTED H_OnResetting : E_PackMLHookResult
VAR_INPUT
	bFirstScan	: BOOL;
END_VAR
H_OnResetting := E_PackMLHookResult.Done;
END_METHOD

METHOD PROTECTED H_OnStarting : E_PackMLHookResult
VAR_INPUT
	bFirstScan	: BOOL;
END_VAR
H_OnStarting := E_PackMLHookResult.Busy;

// Validate Service-owned data before reserving the shared BaseUnit.
IF Param.Velocity <= 0 THEN
	M_AddError(MainErrorId := E_Chamber1ErrorCode.Invalid_Param, SourceErrorId := 0, Message := 'Velocity must be greater than zero.');
	RequestCommand(E_PackMLCommand.Abort);
	RETURN;
END_IF

IF Param.Acceleration < 0 THEN
	M_AddError(MainErrorId := E_Chamber1ErrorCode.Invalid_Param, SourceErrorId := 0, Message := 'Acceleration must not be negative.');
	RequestCommand(E_PackMLCommand.Abort);
	RETURN;
END_IF

IF Param.Deceleration < 0 THEN
	M_AddError(MainErrorId := E_Chamber1ErrorCode.Invalid_Param, SourceErrorId := 0, Message := 'Deceleration must not be negative.');
	RequestCommand(E_PackMLCommand.Abort);
	RETURN;
END_IF

// Resource contention is a failed Start, not a wait condition.
IF NOT Axis_BaseUnit.M_AcquireResource(OwnerId := ServiceId) THEN
	M_AddError(MainErrorId := E_Chamber1ErrorCode.Resource_Acquire_Failed_During_Starting, SourceErrorId := 0, Message := 'Axis resource acquisition failed during Starting.');
	RequestCommand(E_PackMLCommand.Abort);
	RETURN;
END_IF

// Physical checks occur only after this Service owns the BaseUnit.
IF Axis_BaseUnit.AxisIsDisabled THEN
	M_AddError(MainErrorId := E_Chamber1ErrorCode.Axis_Not_Servo_On_During_Starting, SourceErrorId := 0, Message := 'Axis is not servo on during Starting.');
	RequestCommand(E_PackMLCommand.Abort);
	RETURN;
END_IF

IF Axis_BaseUnit.AxisHasJob THEN
	M_AddError(MainErrorId := E_Chamber1ErrorCode.Axis_Is_Busy_During_Starting, SourceErrorId := 0, Message := 'Axis is busy during Starting.');
	RequestCommand(E_PackMLCommand.Abort);
	RETURN;
END_IF

H_OnStarting := E_PackMLHookResult.Done;
END_METHOD

METHOD PROTECTED H_OnStopped
VAR_INPUT
	bFirstScan	: BOOL;
END_VAR
// Release defensively after every Stop path.
Axis_BaseUnit.M_ReleaseResource(OwnerId := ServiceId);
END_METHOD

METHOD PROTECTED H_OnStopping : E_PackMLHookResult
VAR_INPUT
	bFirstScan	: BOOL;
END_VAR
H_OnStopping := E_PackMLHookResult.Done;

// Resource acquisition failures enter Stopping without owning the Axis.
IF NOT Axis_BaseUnit.M_IsResourceOwner(OwnerId := ServiceId) THEN
	RETURN;
END_IF

Axis_BaseUnit.M_Jog(
	OwnerId:= ServiceId,
	JogForward:= FALSE, 
	JogBackwards:= FALSE, 
	Mode:= E_JogMode.MC_JOGMODE_CONTINOUS,
	Position:= Param.Position,
	Velocity:= Param.Velocity,
	Acceleration:= Param.Acceleration,
	Deceleration:= Param.Deceleration);

// Jog is stopped once both direction commands have been withdrawn.
Axis_BaseUnit.M_ReleaseResource(OwnerId := ServiceId);
END_METHOD

END_FUNCTION_BLOCK

// ---- POUs/10_Chamber1/Services/SpinAxis/FB_Chamber1SpinAxisMoveAbsServices.TcPOU
FUNCTION_BLOCK FB_Chamber1SpinAxisMoveAbsServices EXTENDS FB_ServiceBase
VAR_INPUT
	Param : ST_Chamber1SpinAxisMoveAbsParam;
	Axis_BaseUnit : I_Axis_BaseUnit;
END_VAR

M_UpdateService(CompletionBehavior := E_ServiceCompletionBehavior.NaturalCompletion);

METHOD PROTECTED H_OnAborted
VAR_INPUT
	bFirstScan	: BOOL;
END_VAR
// Release defensively in case an unexpected transition skipped cleanup.
Axis_BaseUnit.M_ReleaseResource(OwnerId := ServiceId);
END_METHOD

METHOD PROTECTED H_OnAborting : E_PackMLHookResult
VAR_INPUT
	bFirstScan	: BOOL;
END_VAR

VAR
	bDone : BOOL;
	bError : BOOL;
	nErrorId : UDINT;
END_VAR
H_OnAborting := E_PackMLHookResult.Busy;

// A Service that never acquired the Resource must not reset its Owner's Axis.
IF NOT Axis_BaseUnit.M_IsResourceOwner(OwnerId := ServiceId) THEN
	H_OnAborting := E_PackMLHookResult.Done;
	RETURN;
END_IF

// Withdraw MoveAbsolute before resetting the Axis.
Axis_BaseUnit.M_MoveAbs(
	OwnerId := ServiceId,
	Execute := FALSE,
	Position:= Param.Position,
	Velocity:= Param.Velocity,
	Acceleration:= Param.Acceleration,
	Deceleration:= Param.Deceleration);
	
Axis_BaseUnit.M_Reset(
	OwnerId := ServiceId,
	Execute := TRUE,
	Done=> bDone, Error=> bError, ErrorId=> nErrorId);

IF bDone THEN
	Axis_BaseUnit.M_Reset(
		OwnerId := ServiceId,
		Execute := FALSE);
	// Keep ownership until the asynchronous Reset has completed.
	Axis_BaseUnit.M_ReleaseResource(OwnerId := ServiceId);
	H_OnAborting := E_PackMLHookResult.Done;

ELSIF bError THEN
	// A failed Reset is terminal for this Abort sequence; do not remain in Aborting.
	Axis_BaseUnit.M_Reset(
		OwnerId := ServiceId,
		Execute := FALSE);
	M_AddError(
		MainErrorId := E_Chamber1ErrorCode.Error_While_Reset_Axis,
		SourceErrorId := nErrorId,
		Message := 'Axis reset failed while aborting.');
	Axis_BaseUnit.M_ReleaseResource(OwnerId := ServiceId);
	H_OnAborting := E_PackMLHookResult.Done;
END_IF
END_METHOD

METHOD PROTECTED H_OnClearing : E_PackMLHookResult
VAR_INPUT
	bFirstScan	: BOOL;
END_VAR
M_ClearAllError();
H_OnClearing := E_PackMLHookResult.Done;
END_METHOD

METHOD PROTECTED H_OnComplete
VAR_INPUT
	bFirstScan	: BOOL;
END_VAR
// Completing normally releases first; this is an idempotent safety net.
Axis_BaseUnit.M_ReleaseResource(OwnerId := ServiceId);
END_METHOD

METHOD PROTECTED H_OnCompleting : E_PackMLHookResult
VAR_INPUT
	bFirstScan	: BOOL;
END_VAR
Axis_BaseUnit.M_MoveAbs(
	OwnerId:= ServiceId,
	Execute:= FALSE,
	Position:= Param.Position,
	Velocity:= Param.Velocity,
	Acceleration:= Param.Acceleration,
	Deceleration:= Param.Deceleration);

// Release only after the active MoveAbsolute request has been withdrawn.
Axis_BaseUnit.M_ReleaseResource(OwnerId := ServiceId);
H_OnCompleting := E_PackMLHookResult.Done;
END_METHOD

METHOD PROTECTED H_OnExecute : E_PackMLHookResult
VAR_INPUT
	bFirstScan	: BOOL;
END_VAR

VAR
	bDone : BOOL;
	bError : BOOL;
	nErrorId : UDINT;
END_VAR
H_OnExecute := E_PackMLHookResult.Busy;

Axis_BaseUnit.M_MoveAbs(
	OwnerId:= ServiceId,
	Execute:= TRUE,
	Position:= Param.Position,
	Velocity:= Param.Velocity,
	Acceleration:= Param.Acceleration,
	Deceleration:= Param.Deceleration,
	Done=> bDone, Error=> bError, ErrorId=> nErrorId);


IF bDone THEN
	H_OnExecute := E_PackMLHookResult.Done;
	RETURN;
END_IF

IF bError THEN
	M_AddError(
		MainErrorId := E_Chamber1ErrorCode.Axis_Command_Error_During_Execute,
		SourceErrorId := nErrorId,
		Message := 'MoveAbsolute failed during Execute.');
	RequestCommand(E_PackMLCommand.Abort);
END_IF
END_METHOD

METHOD PROTECTED H_OnIdle
VAR_INPUT
	bFirstScan	: BOOL;
END_VAR
// Idle Services must not retain a Resource from an earlier operation.
Axis_BaseUnit.M_ReleaseResource(OwnerId := ServiceId);
END_METHOD

METHOD PROTECTED H_OnResetting : E_PackMLHookResult
VAR_INPUT
	bFirstScan	: BOOL;
END_VAR
H_OnResetting := E_PackMLHookResult.Done;
END_METHOD

METHOD PROTECTED H_OnStarting : E_PackMLHookResult
VAR_INPUT
	bFirstScan	: BOOL;
END_VAR
H_OnStarting := E_PackMLHookResult.Busy;

// Validate Service-owned data before reserving the shared BaseUnit.
IF Param.Velocity <= 0 THEN
	M_AddError(MainErrorId := E_Chamber1ErrorCode.Invalid_Param, SourceErrorId := 0, Message := 'Velocity must be greater than zero.');
	RequestCommand(E_PackMLCommand.Abort);
	RETURN;
END_IF

IF Param.Acceleration < 0 THEN
	M_AddError(MainErrorId := E_Chamber1ErrorCode.Invalid_Param, SourceErrorId := 0, Message := 'Acceleration must not be negative.');
	RequestCommand(E_PackMLCommand.Abort);
	RETURN;
END_IF

IF Param.Deceleration < 0 THEN
	M_AddError(MainErrorId := E_Chamber1ErrorCode.Invalid_Param, SourceErrorId := 0, Message := 'Deceleration must not be negative.');
	RequestCommand(E_PackMLCommand.Abort);
	RETURN;
END_IF

// Resource contention is a failed Start, not a wait condition.
IF NOT Axis_BaseUnit.M_AcquireResource(OwnerId := ServiceId) THEN
	M_AddError(MainErrorId := E_Chamber1ErrorCode.Resource_Acquire_Failed_During_Starting, SourceErrorId := 0, Message := 'Axis resource acquisition failed during Starting.');
	RequestCommand(E_PackMLCommand.Abort);
	RETURN;
END_IF

// Physical checks occur only after this Service owns the BaseUnit.
IF Axis_BaseUnit.AxisIsDisabled THEN
	M_AddError(MainErrorId := E_Chamber1ErrorCode.Axis_Not_Servo_On_During_Starting, SourceErrorId := 0, Message := 'Axis is not servo on during Starting.');
	RequestCommand(E_PackMLCommand.Abort);
	RETURN;
END_IF

IF Axis_BaseUnit.AxisHasJob THEN
	M_AddError(MainErrorId := E_Chamber1ErrorCode.Axis_Is_Busy_During_Starting, SourceErrorId := 0, Message := 'Axis is busy during Starting.');
	RequestCommand(E_PackMLCommand.Abort);
	RETURN;
END_IF

H_OnStarting := E_PackMLHookResult.Done;
END_METHOD

METHOD PROTECTED H_OnStopped
VAR_INPUT
	bFirstScan	: BOOL;
END_VAR
// Release defensively after every Stop path.
Axis_BaseUnit.M_ReleaseResource(OwnerId := ServiceId);
END_METHOD

METHOD PROTECTED H_OnStopping : E_PackMLHookResult
VAR_INPUT
	bFirstScan	: BOOL;
END_VAR

VAR
	bDone : BOOL;
	bError : BOOL;
	nErrorId : UDINT;
END_VAR
H_OnStopping := E_PackMLHookResult.Busy;

// Resource acquisition failures enter Stopping without owning the Axis.
IF NOT Axis_BaseUnit.M_IsResourceOwner(OwnerId := ServiceId) THEN
	H_OnStopping := E_PackMLHookResult.Done;
	RETURN;
END_IF

// Withdraw MoveAbsolute before issuing the physical Stop.
Axis_BaseUnit.M_MoveAbs(
	OwnerId := ServiceId,
	Execute := FALSE,
	Position:= Param.Position,
	Velocity:= Param.Velocity,
	Acceleration:= Param.Acceleration,
	Deceleration:= Param.Deceleration);
	
Axis_BaseUnit.M_Stop(
	OwnerId := ServiceId,
	Execute := TRUE, 
	Deceleration:= Param.Deceleration,
	Done=> bDone, Error=> bError, ErrorId=> nErrorId);

IF bDone THEN
	Axis_BaseUnit.M_Stop(
		OwnerId := ServiceId,
		Execute := FALSE, 
		Deceleration:= Param.Deceleration);
	// Ownership is released only after the asynchronous Stop has completed.
	Axis_BaseUnit.M_ReleaseResource(OwnerId := ServiceId);
	H_OnStopping := E_PackMLHookResult.Done;
	
ELSIF bError THEN
	// Throw up error
	M_AddError(
		MainErrorId := E_Chamber1ErrorCode.Error_While_Stop_Axis,
		SourceErrorId := nErrorId,
		Message := 'Axis stop failed while stopping.');
	
	Axis_BaseUnit.M_Stop(
		OwnerId := ServiceId,
		Execute := FALSE, 
		Deceleration:= Param.Deceleration);
		
	RequestCommand(E_PackMLCommand.Abort);
END_IF
END_METHOD

END_FUNCTION_BLOCK

// ---- POUs/10_Chamber1/Services/SpinAxis/FB_Chamber1SpinAxisMoveVelCWServices.TcPOU
FUNCTION_BLOCK FB_Chamber1SpinAxisMoveVelCWServices EXTENDS FB_ServiceBase
VAR_INPUT
	Param : ST_Chamber1SpinAxisMoveVelParam;
	Axis_BaseUnit : I_Axis_BaseUnit;
END_VAR

VAR
	_LatchedParam : ST_Chamber1SpinAxisMoveVelParam;
END_VAR

M_UpdateService(CompletionBehavior := E_ServiceCompletionBehavior.NaturalCompletion);

METHOD PROTECTED H_OnAborted
VAR_INPUT
	bFirstScan	: BOOL;
END_VAR
// Release defensively in case an unexpected transition skipped cleanup.
Axis_BaseUnit.M_ReleaseResource(OwnerId := ServiceId);
END_METHOD

METHOD PROTECTED H_OnAborting : E_PackMLHookResult
VAR_INPUT
	bFirstScan	: BOOL;
END_VAR

VAR
	bDone : BOOL;
	bError : BOOL;
	nErrorId : UDINT;
END_VAR
H_OnAborting := E_PackMLHookResult.Busy;

// A Service that never acquired the Resource must not reset its Owner's Axis.
IF NOT Axis_BaseUnit.M_IsResourceOwner(OwnerId := ServiceId) THEN
	H_OnAborting := E_PackMLHookResult.Done;
	RETURN;
END_IF

// Withdraw MoveVelocity before resetting the Axis.
Axis_BaseUnit.M_MoveVel(
	OwnerId := ServiceId,
	Execute := FALSE,
	Direction := MC_Direction.MC_Positive_Direction,
	Velocity := _LatchedParam.Velocity,
	Acceleration := _LatchedParam.Acceleration,
	Deceleration := _LatchedParam.Deceleration);
	
Axis_BaseUnit.M_Reset(
	OwnerId := ServiceId,
	Execute := TRUE,
	Done=> bDone, Error=> bError, ErrorId=> nErrorId);

IF bDone THEN
	Axis_BaseUnit.M_Reset(
		OwnerId := ServiceId,
		Execute := FALSE);
	// Keep ownership until the asynchronous Reset has completed.
	Axis_BaseUnit.M_ReleaseResource(OwnerId := ServiceId);
	H_OnAborting := E_PackMLHookResult.Done;

ELSIF bError THEN
	// A failed Reset is terminal for this Abort sequence; do not remain in Aborting.
	Axis_BaseUnit.M_Reset(
		OwnerId := ServiceId,
		Execute := FALSE);
	M_AddError(
		MainErrorId := E_Chamber1ErrorCode.Error_While_Reset_Axis,
		SourceErrorId := nErrorId,
		Message := 'Axis reset failed while aborting.');
	Axis_BaseUnit.M_ReleaseResource(OwnerId := ServiceId);
	H_OnAborting := E_PackMLHookResult.Done;
END_IF
END_METHOD

METHOD PROTECTED H_OnClearing : E_PackMLHookResult
VAR_INPUT
	bFirstScan	: BOOL;
END_VAR
M_ClearAllError();
H_OnClearing := E_PackMLHookResult.Done;
END_METHOD

METHOD PROTECTED H_OnComplete
VAR_INPUT
	bFirstScan	: BOOL;
END_VAR
// Reaching Complete means target velocity was reached; the Axis is still moving,
// so this Service must retain ownership until Stop or Abort cleanup finishes.
END_METHOD

METHOD PROTECTED H_OnCompleting : E_PackMLHookResult
VAR_INPUT
	bFirstScan	: BOOL;
END_VAR
Axis_BaseUnit.M_MoveVel(
	OwnerId := ServiceId,
	Execute := FALSE,
	Direction := MC_Direction.MC_Positive_Direction,
	Velocity := _LatchedParam.Velocity,
	Acceleration := _LatchedParam.Acceleration,
	Deceleration := _LatchedParam.Deceleration);

// Lowering Execute only withdraws the FB request; it does not stop the Axis.
// Keep ownership so a later Stop from Complete or Idle can control the motion.
H_OnCompleting := E_PackMLHookResult.Done;
END_METHOD

METHOD PROTECTED H_OnExecute : E_PackMLHookResult
VAR_INPUT
	bFirstScan	: BOOL;
END_VAR

VAR
	bInVelocity : BOOL;
	bError : BOOL;
END_VAR
H_OnExecute := E_PackMLHookResult.Busy;

// The Start-time snapshot remains fixed for the entire Execute phase.
Axis_BaseUnit.M_MoveVel(
	OwnerId := ServiceId,
	Execute := TRUE,
	Direction := MC_Direction.MC_Positive_Direction,
	Velocity := _LatchedParam.Velocity,
	Acceleration := _LatchedParam.Acceleration,
	Deceleration := _LatchedParam.Deceleration,
	InVelocity => bInVelocity,
	Error => bError);

IF bError THEN
	M_AddError(MainErrorId := E_Chamber1ErrorCode.Axis_Command_Error_During_Execute, SourceErrorId := 0, Message := 'MoveVelocity failed during Execute.');
	RequestCommand(E_PackMLCommand.Abort);
	RETURN;
END_IF

IF bInVelocity THEN
	H_OnExecute := E_PackMLHookResult.Done;
END_IF
END_METHOD

METHOD PROTECTED H_OnIdle
VAR_INPUT
	bFirstScan	: BOOL;
END_VAR
// Reset changes only the PackML state. A MoveVel that completed naturally may
// still be moving, so Idle intentionally retains any existing Axis ownership.
END_METHOD

METHOD PROTECTED H_OnResetting : E_PackMLHookResult
VAR_INPUT
	bFirstScan	: BOOL;
END_VAR
H_OnResetting := E_PackMLHookResult.Done;
END_METHOD

METHOD PROTECTED H_OnStarting : E_PackMLHookResult
VAR_INPUT
	bFirstScan	: BOOL;
END_VAR
H_OnStarting := E_PackMLHookResult.Busy;

// Validate Service-owned data before reserving the shared BaseUnit.
IF Param.Velocity <= 0 THEN
	M_AddError(MainErrorId := E_Chamber1ErrorCode.Invalid_Param, SourceErrorId := 0, Message := 'Velocity must be greater than zero.');
	RequestCommand(E_PackMLCommand.Abort);
	RETURN;
END_IF

IF Param.Acceleration < 0 THEN
	M_AddError(MainErrorId := E_Chamber1ErrorCode.Invalid_Param, SourceErrorId := 0, Message := 'Acceleration must not be negative.');
	RequestCommand(E_PackMLCommand.Abort);
	RETURN;
END_IF

IF Param.Deceleration < 0 THEN
	M_AddError(MainErrorId := E_Chamber1ErrorCode.Invalid_Param, SourceErrorId := 0, Message := 'Deceleration must not be negative.');
	RequestCommand(E_PackMLCommand.Abort);
	RETURN;
END_IF

// Keep one fixed command snapshot until the Service leaves this run.
_LatchedParam := Param;

// Resource contention is a failed Start, not a wait condition.
IF NOT Axis_BaseUnit.M_AcquireResource(OwnerId := ServiceId) THEN
	M_AddError(MainErrorId := E_Chamber1ErrorCode.Resource_Acquire_Failed_During_Starting, SourceErrorId := 0, Message := 'Axis resource acquisition failed during Starting.');
	RequestCommand(E_PackMLCommand.Abort);
	RETURN;
END_IF

// Physical checks occur only after this Service owns the BaseUnit.
IF Axis_BaseUnit.AxisIsDisabled THEN
	M_AddError(MainErrorId := E_Chamber1ErrorCode.Axis_Not_Servo_On_During_Starting, SourceErrorId := 0, Message := 'Axis is not servo on during Starting.');
	RequestCommand(E_PackMLCommand.Abort);
	RETURN;
END_IF

IF Axis_BaseUnit.AxisHasJob THEN
	M_AddError(MainErrorId := E_Chamber1ErrorCode.Axis_Is_Busy_During_Starting, SourceErrorId := 0, Message := 'Axis is busy during Starting.');
	RequestCommand(E_PackMLCommand.Abort);
	RETURN;
END_IF

H_OnStarting := E_PackMLHookResult.Done;
END_METHOD

METHOD PROTECTED H_OnStopped
VAR_INPUT
	bFirstScan	: BOOL;
END_VAR
// Release defensively after every Stop path.
Axis_BaseUnit.M_ReleaseResource(OwnerId := ServiceId);
END_METHOD

METHOD PROTECTED H_OnStopping : E_PackMLHookResult
VAR_INPUT
	bFirstScan	: BOOL;
END_VAR

VAR
	bDone : BOOL;
	bError : BOOL;
	nErrorId : UDINT;
END_VAR
H_OnStopping := E_PackMLHookResult.Busy;

// Resource acquisition failures enter Stopping without owning the Axis.
IF NOT Axis_BaseUnit.M_IsResourceOwner(OwnerId := ServiceId) THEN
	H_OnStopping := E_PackMLHookResult.Done;
	RETURN;
END_IF

// Withdraw MoveVelocity before issuing the physical Stop.
Axis_BaseUnit.M_MoveVel(
	OwnerId := ServiceId,
	Execute := FALSE,
	Direction := MC_Direction.MC_Positive_Direction,
	Velocity := _LatchedParam.Velocity,
	Acceleration := _LatchedParam.Acceleration,
	Deceleration := _LatchedParam.Deceleration);
	
Axis_BaseUnit.M_Stop(
	OwnerId := ServiceId,
	Execute := TRUE, 
	Deceleration:= _LatchedParam.Deceleration,
	Done=> bDone, Error=> bError, ErrorId=> nErrorId);

IF bDone THEN
	Axis_BaseUnit.M_Stop(
		OwnerId := ServiceId,
		Execute := FALSE, 
		Deceleration:= _LatchedParam.Deceleration);
	// Ownership is released only after the asynchronous Stop has completed.
	Axis_BaseUnit.M_ReleaseResource(OwnerId := ServiceId);
	H_OnStopping := E_PackMLHookResult.Done;
	
ELSIF bError THEN
	// Throw up error
	M_AddError(
		MainErrorId := E_Chamber1ErrorCode.Error_While_Stop_Axis,
		SourceErrorId := nErrorId,
		Message := 'Axis stop failed while stopping.');
	
	Axis_BaseUnit.M_Stop(
		OwnerId := ServiceId,
		Execute := FALSE, 
		Deceleration:= _LatchedParam.Deceleration);
		
	RequestCommand(E_PackMLCommand.Abort);
END_IF
END_METHOD

END_FUNCTION_BLOCK

// ---- POUs/10_Chamber1/Services/LiftAxis/FB_Chamber1LiftPinAxisMoveVelCWServices.TcPOU
FUNCTION_BLOCK FB_Chamber1LiftPinAxisMoveVelCWServices EXTENDS FB_ServiceBase
VAR_INPUT
	Param : ST_Chamber1LiftPinAxisMoveVelParam;
	Axis_BaseUnit : I_Axis_BaseUnit;
END_VAR

VAR
	_LatchedParam : ST_Chamber1LiftPinAxisMoveVelParam;
END_VAR

M_UpdateService(CompletionBehavior := E_ServiceCompletionBehavior.NaturalCompletion);

METHOD PROTECTED H_OnAborted
VAR_INPUT
	bFirstScan	: BOOL;
END_VAR
// Release defensively in case an unexpected transition skipped cleanup.
Axis_BaseUnit.M_ReleaseResource(OwnerId := ServiceId);
END_METHOD

METHOD PROTECTED H_OnAborting : E_PackMLHookResult
VAR_INPUT
	bFirstScan	: BOOL;
END_VAR

VAR
	bDone : BOOL;
	bError : BOOL;
	nErrorId : UDINT;
END_VAR
H_OnAborting := E_PackMLHookResult.Busy;

// A Service that never acquired the Resource must not reset its Owner's Axis.
IF NOT Axis_BaseUnit.M_IsResourceOwner(OwnerId := ServiceId) THEN
	H_OnAborting := E_PackMLHookResult.Done;
	RETURN;
END_IF

// Withdraw MoveVelocity before resetting the Axis.
Axis_BaseUnit.M_MoveVel(
	OwnerId := ServiceId,
	Execute := FALSE,
	Direction := MC_Direction.MC_Positive_Direction,
	Velocity := _LatchedParam.Velocity,
	Acceleration := _LatchedParam.Acceleration,
	Deceleration := _LatchedParam.Deceleration);

Axis_BaseUnit.M_Reset(
	OwnerId := ServiceId,
	Execute := TRUE,
	Done=> bDone, Error=> bError, ErrorId=> nErrorId);

IF bDone THEN
	Axis_BaseUnit.M_Reset(
		OwnerId := ServiceId,
		Execute := FALSE);
	// Keep ownership until the asynchronous Reset has completed.
	Axis_BaseUnit.M_ReleaseResource(OwnerId := ServiceId);
	H_OnAborting := E_PackMLHookResult.Done;

ELSIF bError THEN
	// A failed Reset is terminal for this Abort sequence; do not remain in Aborting.
	Axis_BaseUnit.M_Reset(
		OwnerId := ServiceId,
		Execute := FALSE);
	M_AddError(
		MainErrorId := E_Chamber1ErrorCode.Error_While_Reset_Axis,
		SourceErrorId := nErrorId,
		Message := 'Axis reset failed while aborting.');
	Axis_BaseUnit.M_ReleaseResource(OwnerId := ServiceId);
	H_OnAborting := E_PackMLHookResult.Done;
END_IF
END_METHOD

METHOD PROTECTED H_OnClearing : E_PackMLHookResult
VAR_INPUT
	bFirstScan	: BOOL;
END_VAR
M_ClearAllError();
H_OnClearing := E_PackMLHookResult.Done;
END_METHOD

METHOD PROTECTED H_OnComplete
VAR_INPUT
	bFirstScan	: BOOL;
END_VAR
// Reaching Complete means target velocity was reached; the Axis is still moving,
// so this Service must retain ownership until Stop or Abort cleanup finishes.
END_METHOD

METHOD PROTECTED H_OnCompleting : E_PackMLHookResult
VAR_INPUT
	bFirstScan	: BOOL;
END_VAR
Axis_BaseUnit.M_MoveVel(
	OwnerId := ServiceId,
	Execute := FALSE,
	Direction := MC_Direction.MC_Positive_Direction,
	Velocity := _LatchedParam.Velocity,
	Acceleration := _LatchedParam.Acceleration,
	Deceleration := _LatchedParam.Deceleration);

// Lowering Execute only withdraws the FB request; it does not stop the Axis.
// Keep ownership so a later Stop from Complete or Idle can control the motion.
H_OnCompleting := E_PackMLHookResult.Done;
END_METHOD

METHOD PROTECTED H_OnExecute : E_PackMLHookResult
VAR_INPUT
	bFirstScan	: BOOL;
END_VAR

VAR
	bInVelocity : BOOL;
	bError : BOOL;
END_VAR
H_OnExecute := E_PackMLHookResult.Busy;

// The Start-time snapshot remains fixed for the entire Execute phase.
Axis_BaseUnit.M_MoveVel(
	OwnerId := ServiceId,
	Execute := TRUE,
	Direction := MC_Direction.MC_Positive_Direction,
	Velocity := _LatchedParam.Velocity,
	Acceleration := _LatchedParam.Acceleration,
	Deceleration := _LatchedParam.Deceleration,
	InVelocity => bInVelocity,
	Error => bError);

IF bError THEN
	M_AddError(MainErrorId := E_Chamber1ErrorCode.Axis_Command_Error_During_Execute, SourceErrorId := 0, Message := 'MoveVelocity failed during Execute.');
	RequestCommand(E_PackMLCommand.Abort);
	RETURN;
END_IF

IF bInVelocity THEN
	H_OnExecute := E_PackMLHookResult.Done;
END_IF
END_METHOD

METHOD PROTECTED H_OnIdle
VAR_INPUT
	bFirstScan	: BOOL;
END_VAR
// Reset changes only the PackML state. A MoveVel that completed naturally may
// still be moving, so Idle intentionally retains any existing Axis ownership.
END_METHOD

METHOD PROTECTED H_OnResetting : E_PackMLHookResult
VAR_INPUT
	bFirstScan	: BOOL;
END_VAR
H_OnResetting := E_PackMLHookResult.Done;
END_METHOD

METHOD PROTECTED H_OnStarting : E_PackMLHookResult
VAR_INPUT
	bFirstScan	: BOOL;
END_VAR
H_OnStarting := E_PackMLHookResult.Busy;

// Validate Service-owned data before reserving the shared BaseUnit.
IF Param.Velocity <= 0 THEN
	M_AddError(MainErrorId := E_Chamber1ErrorCode.Invalid_Param, SourceErrorId := 0, Message := 'Velocity must be greater than zero.');
	RequestCommand(E_PackMLCommand.Abort);
	RETURN;
END_IF

IF Param.Acceleration < 0 THEN
	M_AddError(MainErrorId := E_Chamber1ErrorCode.Invalid_Param, SourceErrorId := 0, Message := 'Acceleration must not be negative.');
	RequestCommand(E_PackMLCommand.Abort);
	RETURN;
END_IF

IF Param.Deceleration < 0 THEN
	M_AddError(MainErrorId := E_Chamber1ErrorCode.Invalid_Param, SourceErrorId := 0, Message := 'Deceleration must not be negative.');
	RequestCommand(E_PackMLCommand.Abort);
	RETURN;
END_IF

// Keep one fixed command snapshot until the Service leaves this run.
_LatchedParam := Param;

// Resource contention is a failed Start, not a wait condition.
IF NOT Axis_BaseUnit.M_AcquireResource(OwnerId := ServiceId) THEN
	M_AddError(MainErrorId := E_Chamber1ErrorCode.Resource_Acquire_Failed_During_Starting, SourceErrorId := 0, Message := 'Axis resource acquisition failed during Starting.');
	RequestCommand(E_PackMLCommand.Abort);
	RETURN;
END_IF

// Physical checks occur only after this Service owns the BaseUnit.
IF Axis_BaseUnit.AxisIsDisabled THEN
	M_AddError(MainErrorId := E_Chamber1ErrorCode.Axis_Not_Servo_On_During_Starting, SourceErrorId := 0, Message := 'Axis is not servo on during Starting.');
	RequestCommand(E_PackMLCommand.Abort);
	RETURN;
END_IF

IF Axis_BaseUnit.AxisHasJob THEN
	M_AddError(MainErrorId := E_Chamber1ErrorCode.Axis_Is_Busy_During_Starting, SourceErrorId := 0, Message := 'Axis is busy during Starting.');
	RequestCommand(E_PackMLCommand.Abort);
	RETURN;
END_IF

H_OnStarting := E_PackMLHookResult.Done;
END_METHOD

METHOD PROTECTED H_OnStopped
VAR_INPUT
	bFirstScan	: BOOL;
END_VAR
// Release defensively after every Stop path.
Axis_BaseUnit.M_ReleaseResource(OwnerId := ServiceId);
END_METHOD

METHOD PROTECTED H_OnStopping : E_PackMLHookResult
VAR_INPUT
	bFirstScan	: BOOL;
END_VAR

VAR
	bDone : BOOL;
	bError : BOOL;
	nErrorId : UDINT;
END_VAR
H_OnStopping := E_PackMLHookResult.Busy;

// Resource acquisition failures enter Stopping without owning the Axis.
IF NOT Axis_BaseUnit.M_IsResourceOwner(OwnerId := ServiceId) THEN
	H_OnStopping := E_PackMLHookResult.Done;
	RETURN;
END_IF

// Withdraw MoveVelocity before issuing the physical Stop.
Axis_BaseUnit.M_MoveVel(
	OwnerId := ServiceId,
	Execute := FALSE,
	Direction := MC_Direction.MC_Positive_Direction,
	Velocity := _LatchedParam.Velocity,
	Acceleration := _LatchedParam.Acceleration,
	Deceleration := _LatchedParam.Deceleration);

Axis_BaseUnit.M_Stop(
	OwnerId := ServiceId,
	Execute := TRUE,
	Deceleration:= _LatchedParam.Deceleration,
	Done=> bDone, Error=> bError, ErrorId=> nErrorId);

IF bDone THEN
	Axis_BaseUnit.M_Stop(
		OwnerId := ServiceId,
		Execute := FALSE,
		Deceleration:= _LatchedParam.Deceleration);
	// Ownership is released only after the asynchronous Stop has completed.
	Axis_BaseUnit.M_ReleaseResource(OwnerId := ServiceId);
	H_OnStopping := E_PackMLHookResult.Done;

ELSIF bError THEN
	// Throw up error
	M_AddError(
		MainErrorId := E_Chamber1ErrorCode.Error_While_Stop_Axis,
		SourceErrorId := nErrorId,
		Message := 'Axis stop failed while stopping.');

	Axis_BaseUnit.M_Stop(
		OwnerId := ServiceId,
		Execute := FALSE,
		Deceleration:= _LatchedParam.Deceleration);

	RequestCommand(E_PackMLCommand.Abort);
END_IF
END_METHOD

END_FUNCTION_BLOCK

// ---- POUs/10_Chamber1/Services/LiftAxis/FB_Chamber1LiftPinAxisMoveVelCCWServices.TcPOU
FUNCTION_BLOCK FB_Chamber1LiftPinAxisMoveVelCCWServices EXTENDS FB_ServiceBase
VAR_INPUT
	Param : ST_Chamber1LiftPinAxisMoveVelParam;
	Axis_BaseUnit : I_Axis_BaseUnit;
END_VAR

VAR
	_LatchedParam : ST_Chamber1LiftPinAxisMoveVelParam;
END_VAR

M_UpdateService(CompletionBehavior := E_ServiceCompletionBehavior.NaturalCompletion);

METHOD PROTECTED H_OnAborted
VAR_INPUT
	bFirstScan	: BOOL;
END_VAR
// Release defensively in case an unexpected transition skipped cleanup.
Axis_BaseUnit.M_ReleaseResource(OwnerId := ServiceId);
END_METHOD

METHOD PROTECTED H_OnAborting : E_PackMLHookResult
VAR_INPUT
	bFirstScan	: BOOL;
END_VAR

VAR
	bDone : BOOL;
	bError : BOOL;
	nErrorId : UDINT;
END_VAR
H_OnAborting := E_PackMLHookResult.Busy;

// A Service that never acquired the Resource must not reset its Owner's Axis.
IF NOT Axis_BaseUnit.M_IsResourceOwner(OwnerId := ServiceId) THEN
	H_OnAborting := E_PackMLHookResult.Done;
	RETURN;
END_IF

// Withdraw MoveVelocity before resetting the Axis.
Axis_BaseUnit.M_MoveVel(
	OwnerId := ServiceId,
	Execute := FALSE,
	Direction := MC_Direction.MC_Negative_Direction,
	Velocity := _LatchedParam.Velocity,
	Acceleration := _LatchedParam.Acceleration,
	Deceleration := _LatchedParam.Deceleration);

Axis_BaseUnit.M_Reset(
	OwnerId := ServiceId,
	Execute := TRUE,
	Done=> bDone, Error=> bError, ErrorId=> nErrorId);

IF bDone THEN
	Axis_BaseUnit.M_Reset(
		OwnerId := ServiceId,
		Execute := FALSE);
	// Keep ownership until the asynchronous Reset has completed.
	Axis_BaseUnit.M_ReleaseResource(OwnerId := ServiceId);
	H_OnAborting := E_PackMLHookResult.Done;

ELSIF bError THEN
	// A failed Reset is terminal for this Abort sequence; do not remain in Aborting.
	Axis_BaseUnit.M_Reset(
		OwnerId := ServiceId,
		Execute := FALSE);
	M_AddError(
		MainErrorId := E_Chamber1ErrorCode.Error_While_Reset_Axis,
		SourceErrorId := nErrorId,
		Message := 'Axis reset failed while aborting.');
	Axis_BaseUnit.M_ReleaseResource(OwnerId := ServiceId);
	H_OnAborting := E_PackMLHookResult.Done;
END_IF
END_METHOD

METHOD PROTECTED H_OnClearing : E_PackMLHookResult
VAR_INPUT
	bFirstScan	: BOOL;
END_VAR

VAR
	bServoOn : BOOL;
	bError : BOOL;
	nErrorId : UDINT;
END_VAR
M_ClearAllError();
H_OnClearing := E_PackMLHookResult.Done;
END_METHOD

METHOD PROTECTED H_OnComplete
VAR_INPUT
	bFirstScan	: BOOL;
END_VAR
// Reaching Complete means target velocity was reached; the Axis is still moving,
// so this Service must retain ownership until Stop or Abort cleanup finishes.
END_METHOD

METHOD PROTECTED H_OnCompleting : E_PackMLHookResult
VAR_INPUT
	bFirstScan	: BOOL;
END_VAR
Axis_BaseUnit.M_MoveVel(
	OwnerId := ServiceId,
	Execute := FALSE,
	Direction := MC_Direction.MC_Negative_Direction,
	Velocity := _LatchedParam.Velocity,
	Acceleration := _LatchedParam.Acceleration,
	Deceleration := _LatchedParam.Deceleration);

// Lowering Execute only withdraws the FB request; it does not stop the Axis.
// Keep ownership so a later Stop from Complete or Idle can control the motion.
H_OnCompleting := E_PackMLHookResult.Done;
END_METHOD

METHOD PROTECTED H_OnExecute : E_PackMLHookResult
VAR_INPUT
	bFirstScan	: BOOL;
END_VAR

VAR
	bInVelocity : BOOL;
	bError : BOOL;
END_VAR
H_OnExecute := E_PackMLHookResult.Busy;

// The Start-time snapshot remains fixed for the entire Execute phase.
Axis_BaseUnit.M_MoveVel(
	OwnerId := ServiceId,
	Execute := TRUE,
	Direction := MC_Direction.MC_Negative_Direction,
	Velocity := _LatchedParam.Velocity,
	Acceleration := _LatchedParam.Acceleration,
	Deceleration := _LatchedParam.Deceleration,
	InVelocity => bInVelocity,
	Error => bError);

IF bError THEN
	M_AddError(MainErrorId := E_Chamber1ErrorCode.Axis_Command_Error_During_Execute, SourceErrorId := 0, Message := 'MoveVelocity failed during Execute.');
	RequestCommand(E_PackMLCommand.Abort);
	RETURN;
END_IF

IF bInVelocity THEN
	H_OnExecute := E_PackMLHookResult.Done;
END_IF
END_METHOD

METHOD PROTECTED H_OnIdle
VAR_INPUT
	bFirstScan	: BOOL;
END_VAR
// Reset changes only the PackML state. A MoveVel that completed naturally may
// still be moving, so Idle intentionally retains any existing Axis ownership.
END_METHOD

METHOD PROTECTED H_OnResetting : E_PackMLHookResult
VAR_INPUT
	bFirstScan	: BOOL;
END_VAR
H_OnResetting := E_PackMLHookResult.Done;
END_METHOD

METHOD PROTECTED H_OnStarting : E_PackMLHookResult
VAR_INPUT
	bFirstScan	: BOOL;
END_VAR
H_OnStarting := E_PackMLHookResult.Busy;

// Validate Service-owned data before reserving the shared BaseUnit.
IF Param.Velocity <= 0 THEN
	M_AddError(MainErrorId := E_Chamber1ErrorCode.Invalid_Param, SourceErrorId := 0, Message := 'Velocity must be greater than zero.');
	RequestCommand(E_PackMLCommand.Abort);
	RETURN;
END_IF

IF Param.Acceleration < 0 THEN
	M_AddError(MainErrorId := E_Chamber1ErrorCode.Invalid_Param, SourceErrorId := 0, Message := 'Acceleration must not be negative.');
	RequestCommand(E_PackMLCommand.Abort);
	RETURN;
END_IF

IF Param.Deceleration < 0 THEN
	M_AddError(MainErrorId := E_Chamber1ErrorCode.Invalid_Param, SourceErrorId := 0, Message := 'Deceleration must not be negative.');
	RequestCommand(E_PackMLCommand.Abort);
	RETURN;
END_IF

// Keep one fixed command snapshot until the Service leaves this run.
_LatchedParam := Param;

// Resource contention is a failed Start, not a wait condition.
IF NOT Axis_BaseUnit.M_AcquireResource(OwnerId := ServiceId) THEN
	M_AddError(MainErrorId := E_Chamber1ErrorCode.Resource_Acquire_Failed_During_Starting, SourceErrorId := 0, Message := 'Axis resource acquisition failed during Starting.');
	RequestCommand(E_PackMLCommand.Abort);
	RETURN;
END_IF

// Physical checks occur only after this Service owns the BaseUnit.
IF Axis_BaseUnit.AxisIsDisabled THEN
	M_AddError(MainErrorId := E_Chamber1ErrorCode.Axis_Not_Servo_On_During_Starting, SourceErrorId := 0, Message := 'Axis is not servo on during Starting.');
	RequestCommand(E_PackMLCommand.Abort);
	RETURN;
END_IF

IF Axis_BaseUnit.AxisHasJob THEN
	M_AddError(MainErrorId := E_Chamber1ErrorCode.Axis_Is_Busy_During_Starting, SourceErrorId := 0, Message := 'Axis is busy during Starting.');
	RequestCommand(E_PackMLCommand.Abort);
	RETURN;
END_IF

H_OnStarting := E_PackMLHookResult.Done;
END_METHOD

METHOD PROTECTED H_OnStopped
VAR_INPUT
	bFirstScan	: BOOL;
END_VAR
// Release defensively after every Stop path.
Axis_BaseUnit.M_ReleaseResource(OwnerId := ServiceId);
END_METHOD

METHOD PROTECTED H_OnStopping : E_PackMLHookResult
VAR_INPUT
	bFirstScan	: BOOL;
END_VAR

VAR
	bDone : BOOL;
	bError : BOOL;
	nErrorId : UDINT;
END_VAR
H_OnStopping := E_PackMLHookResult.Busy;

// Resource acquisition failures enter Stopping without owning the Axis.
IF NOT Axis_BaseUnit.M_IsResourceOwner(OwnerId := ServiceId) THEN
	H_OnStopping := E_PackMLHookResult.Done;
	RETURN;
END_IF

// Withdraw MoveVelocity before issuing the physical Stop.
Axis_BaseUnit.M_MoveVel(
	OwnerId := ServiceId,
	Execute := FALSE,
	Direction := MC_Direction.MC_Negative_Direction,
	Velocity := _LatchedParam.Velocity,
	Acceleration := _LatchedParam.Acceleration,
	Deceleration := _LatchedParam.Deceleration);

Axis_BaseUnit.M_Stop(
	OwnerId := ServiceId,
	Execute := TRUE,
	Deceleration:= _LatchedParam.Deceleration,
	Done=> bDone, Error=> bError, ErrorId=> nErrorId);

IF bDone THEN
	Axis_BaseUnit.M_Stop(
		OwnerId := ServiceId,
		Execute := FALSE,
		Deceleration:= _LatchedParam.Deceleration);
	// Ownership is released only after the asynchronous Stop has completed.
	Axis_BaseUnit.M_ReleaseResource(OwnerId := ServiceId);
	H_OnStopping := E_PackMLHookResult.Done;

ELSIF bError THEN
	// Throw up error
	M_AddError(
		MainErrorId := E_Chamber1ErrorCode.Error_While_Stop_Axis,
		SourceErrorId := nErrorId,
		Message := 'Axis stop failed while stopping.');

	Axis_BaseUnit.M_Stop(
		OwnerId := ServiceId,
		Execute := FALSE,
		Deceleration:= _LatchedParam.Deceleration);

	RequestCommand(E_PackMLCommand.Abort);
END_IF
END_METHOD

END_FUNCTION_BLOCK

// ---- POUs/10_Chamber1/Services/LiftAxis/FB_Chamber1LiftPinAxisMoveAbsServices.TcPOU
FUNCTION_BLOCK FB_Chamber1LiftPinAxisMoveAbsServices EXTENDS FB_ServiceBase
VAR_INPUT
	Param : ST_Chamber1LiftPinAxisMoveAbsParam;
	Axis_BaseUnit : I_Axis_BaseUnit;
END_VAR

M_UpdateService(CompletionBehavior := E_ServiceCompletionBehavior.NaturalCompletion);

METHOD PROTECTED H_OnAborted
VAR_INPUT
	bFirstScan	: BOOL;
END_VAR
// Release defensively in case an unexpected transition skipped cleanup.
Axis_BaseUnit.M_ReleaseResource(OwnerId := ServiceId);
END_METHOD

METHOD PROTECTED H_OnAborting : E_PackMLHookResult
VAR_INPUT
	bFirstScan	: BOOL;
END_VAR

VAR
	bDone : BOOL;
	bError : BOOL;
	nErrorId : UDINT;
END_VAR
H_OnAborting := E_PackMLHookResult.Busy;

// A Service that never acquired the Resource must not reset its Owner's Axis.
IF NOT Axis_BaseUnit.M_IsResourceOwner(OwnerId := ServiceId) THEN
	H_OnAborting := E_PackMLHookResult.Done;
	RETURN;
END_IF

// Withdraw MoveAbsolute before resetting the Axis.
Axis_BaseUnit.M_MoveAbs(
	OwnerId := ServiceId,
	Execute := FALSE,
	Position:= Param.Position,
	Velocity:= Param.Velocity,
	Acceleration:= Param.Acceleration,
	Deceleration:= Param.Deceleration);

Axis_BaseUnit.M_Reset(
	OwnerId := ServiceId,
	Execute := TRUE,
	Done=> bDone, Error=> bError, ErrorId=> nErrorId);

IF bDone THEN
	Axis_BaseUnit.M_Reset(
		OwnerId := ServiceId,
		Execute := FALSE);
	// Keep ownership until the asynchronous Reset has completed.
	Axis_BaseUnit.M_ReleaseResource(OwnerId := ServiceId);
	H_OnAborting := E_PackMLHookResult.Done;

ELSIF bError THEN
	// A failed Reset is terminal for this Abort sequence; do not remain in Aborting.
	Axis_BaseUnit.M_Reset(
		OwnerId := ServiceId,
		Execute := FALSE);
	M_AddError(
		MainErrorId := E_Chamber1ErrorCode.Error_While_Reset_Axis,
		SourceErrorId := nErrorId,
		Message := 'Axis reset failed while aborting.');
	Axis_BaseUnit.M_ReleaseResource(OwnerId := ServiceId);
	H_OnAborting := E_PackMLHookResult.Done;
END_IF
END_METHOD

METHOD PROTECTED H_OnClearing : E_PackMLHookResult
VAR_INPUT
	bFirstScan	: BOOL;
END_VAR

VAR
	bServoOn : BOOL;
	bError : BOOL;
	nErrorId : UDINT;
END_VAR
M_ClearAllError();
H_OnClearing := E_PackMLHookResult.Done;
END_METHOD

METHOD PROTECTED H_OnComplete
VAR_INPUT
	bFirstScan	: BOOL;
END_VAR
// Completing normally releases first; this is an idempotent safety net.
Axis_BaseUnit.M_ReleaseResource(OwnerId := ServiceId);
END_METHOD

METHOD PROTECTED H_OnCompleting : E_PackMLHookResult
VAR_INPUT
	bFirstScan	: BOOL;
END_VAR
Axis_BaseUnit.M_MoveAbs(
	OwnerId:= ServiceId,
	Execute:= FALSE,
	Position:= Param.Position,
	Velocity:= Param.Velocity,
	Acceleration:= Param.Acceleration,
	Deceleration:= Param.Deceleration);

// Release only after the active MoveAbsolute request has been withdrawn.
Axis_BaseUnit.M_ReleaseResource(OwnerId := ServiceId);
H_OnCompleting := E_PackMLHookResult.Done;
END_METHOD

METHOD PROTECTED H_OnExecute : E_PackMLHookResult
VAR_INPUT
	bFirstScan	: BOOL;
END_VAR

VAR
	bDone : BOOL;
	bError : BOOL;
	nErrorId : UDINT;
END_VAR
H_OnExecute := E_PackMLHookResult.Busy;

Axis_BaseUnit.M_MoveAbs(
	OwnerId:= ServiceId,
	Execute:= TRUE,
	Position:= Param.Position,
	Velocity:= Param.Velocity,
	Acceleration:= Param.Acceleration,
	Deceleration:= Param.Deceleration,
	Done=> bDone, Error=> bError, ErrorId=> nErrorId);


IF bDone THEN
	H_OnExecute := E_PackMLHookResult.Done;
	RETURN;
END_IF

IF bError THEN
	M_AddError(
		MainErrorId := E_Chamber1ErrorCode.Axis_Command_Error_During_Execute,
		SourceErrorId := nErrorId,
		Message := 'MoveAbsolute failed during Execute.');
	RequestCommand(E_PackMLCommand.Abort);
END_IF
END_METHOD

METHOD PROTECTED H_OnIdle
VAR_INPUT
	bFirstScan	: BOOL;
END_VAR
// Idle Services must not retain a Resource from an earlier operation.
Axis_BaseUnit.M_ReleaseResource(OwnerId := ServiceId);
END_METHOD

METHOD PROTECTED H_OnResetting : E_PackMLHookResult
VAR_INPUT
	bFirstScan	: BOOL;
END_VAR
H_OnResetting := E_PackMLHookResult.Done;
END_METHOD

METHOD PROTECTED H_OnStarting : E_PackMLHookResult
VAR_INPUT
	bFirstScan	: BOOL;
END_VAR
H_OnStarting := E_PackMLHookResult.Busy;

// Validate Service-owned data before reserving the shared BaseUnit.
IF Param.Velocity <= 0 THEN
	M_AddError(MainErrorId := E_Chamber1ErrorCode.Invalid_Param, SourceErrorId := 0, Message := 'Velocity must be greater than zero.');
	RequestCommand(E_PackMLCommand.Abort);
	RETURN;
END_IF

IF Param.Acceleration < 0 THEN
	M_AddError(MainErrorId := E_Chamber1ErrorCode.Invalid_Param, SourceErrorId := 0, Message := 'Acceleration must not be negative.');
	RequestCommand(E_PackMLCommand.Abort);
	RETURN;
END_IF

IF Param.Deceleration < 0 THEN
	M_AddError(MainErrorId := E_Chamber1ErrorCode.Invalid_Param, SourceErrorId := 0, Message := 'Deceleration must not be negative.');
	RequestCommand(E_PackMLCommand.Abort);
	RETURN;
END_IF

// Resource contention is a failed Start, not a wait condition.
IF NOT Axis_BaseUnit.M_AcquireResource(OwnerId := ServiceId) THEN
	M_AddError(MainErrorId := E_Chamber1ErrorCode.Resource_Acquire_Failed_During_Starting, SourceErrorId := 0, Message := 'Axis resource acquisition failed during Starting.');
	RequestCommand(E_PackMLCommand.Abort);
	RETURN;
END_IF

// Physical checks occur only after this Service owns the BaseUnit.
IF Axis_BaseUnit.AxisIsDisabled THEN
	M_AddError(MainErrorId := E_Chamber1ErrorCode.Axis_Not_Servo_On_During_Starting, SourceErrorId := 0, Message := 'Axis is not servo on during Starting.');
	RequestCommand(E_PackMLCommand.Abort);
	RETURN;
END_IF

IF Axis_BaseUnit.AxisHasJob THEN
	M_AddError(MainErrorId := E_Chamber1ErrorCode.Axis_Is_Busy_During_Starting, SourceErrorId := 0, Message := 'Axis is busy during Starting.');
	RequestCommand(E_PackMLCommand.Abort);
	RETURN;
END_IF

H_OnStarting := E_PackMLHookResult.Done;
END_METHOD

METHOD PROTECTED H_OnStopped
VAR_INPUT
	bFirstScan	: BOOL;
END_VAR
// Release defensively after every Stop path.
Axis_BaseUnit.M_ReleaseResource(OwnerId := ServiceId);
END_METHOD

METHOD PROTECTED H_OnStopping : E_PackMLHookResult
VAR_INPUT
	bFirstScan	: BOOL;
END_VAR

VAR
	bDone : BOOL;
	bError : BOOL;
	nErrorId : UDINT;
END_VAR
H_OnStopping := E_PackMLHookResult.Busy;

// Resource acquisition failures enter Stopping without owning the Axis.
IF NOT Axis_BaseUnit.M_IsResourceOwner(OwnerId := ServiceId) THEN
	H_OnStopping := E_PackMLHookResult.Done;
	RETURN;
END_IF

// Withdraw MoveAbsolute before issuing the physical Stop.
Axis_BaseUnit.M_MoveAbs(
	OwnerId := ServiceId,
	Execute := FALSE,
	Position:= Param.Position,
	Velocity:= Param.Velocity,
	Acceleration:= Param.Acceleration,
	Deceleration:= Param.Deceleration);

Axis_BaseUnit.M_Stop(
	OwnerId := ServiceId,
	Execute := TRUE,
	Deceleration:= Param.Deceleration,
	Done=> bDone, Error=> bError, ErrorId=> nErrorId);

IF bDone THEN
	Axis_BaseUnit.M_Stop(
		OwnerId := ServiceId,
		Execute := FALSE,
		Deceleration:= Param.Deceleration);
	// Ownership is released only after the asynchronous Stop has completed.
	Axis_BaseUnit.M_ReleaseResource(OwnerId := ServiceId);
	H_OnStopping := E_PackMLHookResult.Done;

ELSIF bError THEN
	// Throw up error
	M_AddError(
		MainErrorId := E_Chamber1ErrorCode.Error_While_Stop_Axis,
		SourceErrorId := nErrorId,
		Message := 'Axis stop failed while stopping.');

	Axis_BaseUnit.M_Stop(
		OwnerId := ServiceId,
		Execute := FALSE,
		Deceleration:= Param.Deceleration);

	RequestCommand(E_PackMLCommand.Abort);
END_IF
END_METHOD

END_FUNCTION_BLOCK

// ---- POUs/10_Chamber1/Services/Door/FB_Chamber1Endpoint1DoorOpenService.TcPOU
FUNCTION_BLOCK FB_Chamber1Endpoint1DoorOpenService EXTENDS FB_ServiceBase
VAR_IN_OUT
	IsDoorClose : BOOL;
	DoorCloseCtrl : BOOL;
END_VAR

M_UpdateService(CompletionBehavior := E_ServiceCompletionBehavior.NaturalCompletion);

METHOD PROTECTED H_OnExecute : E_PackMLHookResult
VAR_INPUT
	bFirstScan : BOOL;
END_VAR
H_OnExecute := E_PackMLHookResult.Busy;

DoorCloseCtrl := FALSE;

IF IsDoorClose = FALSE THEN
	H_OnExecute := E_PackMLHookResult.Done;
END_IF
END_METHOD

END_FUNCTION_BLOCK

// ---- POUs/10_Chamber1/Services/Door/FB_Chamber1Endpoint1DoorCloseService.TcPOU
FUNCTION_BLOCK FB_Chamber1Endpoint1DoorCloseService EXTENDS FB_ServiceBase
VAR_IN_OUT
	IsDoorClose : BOOL;
	IsRobotInChamber : BOOL;
	DoorCloseCtrl : BOOL;
END_VAR

M_UpdateService(CompletionBehavior := E_ServiceCompletionBehavior.NaturalCompletion);

METHOD PROTECTED H_OnClearing : RobustSolution_BATW.E_PackMLHookResult
VAR_INPUT
	bFirstScan	: BOOL;
END_VAR
M_ClearAllError();
H_OnClearing := E_PackMLHookResult.Done;
END_METHOD

METHOD PROTECTED H_OnExecute : E_PackMLHookResult
VAR_INPUT
	bFirstScan : BOOL;
END_VAR
H_OnExecute := E_PackMLHookResult.Busy;

DoorCloseCtrl := TRUE;

IF IsDoorClose = TRUE THEN
	H_OnExecute := E_PackMLHookResult.Done;
END_IF
END_METHOD

METHOD PROTECTED H_OnStarting : RobustSolution_BATW.E_PackMLHookResult
VAR_INPUT
	bFirstScan	: BOOL;
END_VAR
H_OnStarting := RobustSolution_BATW.E_PackMLHookResult.Busy;
IF IsRobotInChamber THEN
	M_AddError( MainErrorId:= E_Chamber1ErrorCode.Close_Door_While_Robot_In_Chamber, SourceErrorId:= 0, Message:= 'Close door while robot in chamber.');
	RequestCommand(E_PackMLCommand.Abort);
END_IF

H_OnStarting := RobustSolution_BATW.E_PackMLHookResult.Done;
END_METHOD

END_FUNCTION_BLOCK

// ---- POUs/10_Chamber1/Services/Vacuum/FB_Chamber1VacuumOffService.TcPOU
FUNCTION_BLOCK FB_Chamber1VacuumOffService EXTENDS FB_ServiceBase
VAR_IN_OUT
	IsVacuumOn : BOOL;
	VacuumOnCtrl : BOOL;
END_VAR

M_UpdateService(CompletionBehavior := E_ServiceCompletionBehavior.NaturalCompletion);

METHOD PROTECTED H_OnExecute : E_PackMLHookResult
VAR_INPUT
	bFirstScan : BOOL;
END_VAR
H_OnExecute := E_PackMLHookResult.Busy;

VacuumOnCtrl := FALSE;

IF IsVacuumOn = FALSE THEN
	H_OnExecute := E_PackMLHookResult.Done;
END_IF
END_METHOD

END_FUNCTION_BLOCK

// ---- POUs/10_Chamber1/Services/Vacuum/FB_Chamber1VacuumOnService.TcPOU
FUNCTION_BLOCK FB_Chamber1VacuumOnService EXTENDS FB_ServiceBase
VAR_IN_OUT
	IsVacuumOn : BOOL;
	VacuumOnCtrl : BOOL;
END_VAR

M_UpdateService(CompletionBehavior := E_ServiceCompletionBehavior.NaturalCompletion);

METHOD PROTECTED H_OnExecute : E_PackMLHookResult
VAR_INPUT
	bFirstScan : BOOL;
END_VAR
H_OnExecute := E_PackMLHookResult.Busy;

VacuumOnCtrl := TRUE;

IF IsVacuumOn = TRUE THEN
	H_OnExecute := E_PackMLHookResult.Done;
END_IF
END_METHOD

END_FUNCTION_BLOCK

// ---- POUs/10_Chamber1/Services/FB_Chamber1Ep1PrepareWaferTransfer.TcPOU
FUNCTION_BLOCK FB_Chamber1Ep1PrepareWaferTransfer EXTENDS FB_CompositeServiceBase
VAR
	_Step : E_Ch1Ep1PrepareWaferTransferStep;
	_CommandSubmitted : BOOL;
	_LiftPinMoveParam : ST_Chamber1LiftPinAxisMoveAbsParam;
	_VacuumOffParam : ST_EmptyServiceParam;
END_VAR

M_UpdateCompositeService();

METHOD PROTECTED H_DeclareServices
M_AddDependency(ServiceId := E_Chamber1ServiceId.LiftPinAxisMoveAbs);
M_AddDependency(ServiceId := E_Chamber1ServiceId.VacuumOff);
END_METHOD

METHOD PROTECTED H_GetExecuteSubState : UDINT
H_GetExecuteSubState := TO_UDINT(_Step);
END_METHOD

METHOD PROTECTED H_GetExecuteSubStateName : STRING(80)
H_GetExecuteSubStateName := TO_STRING(_Step);
END_METHOD

METHOD PROTECTED H_OnCompositeExecute : RobustSolution_BATW.E_PackMLHookResult
VAR_INPUT
	bFirstScan	: BOOL;
END_VAR
VAR
	SubmitResult : E_ServiceCallSubmitResult;
	CommandState : E_ServiceInternalCommandState;
	Snapshot : ST_ServiceExecutionSnapshot;
END_VAR
H_OnCompositeExecute := E_PackMLHookResult.Busy;

IF bFirstScan THEN
	_Step := E_Ch1Ep1PrepareWaferTransferStep.MoveLiftPinAxis;
	_CommandSubmitted := FALSE;

	_LiftPinMoveParam.Position := 70.0;
	_LiftPinMoveParam.Velocity := 20.0;
	_LiftPinMoveParam.Acceleration := 0.0;
	_LiftPinMoveParam.Deceleration := 0.0;
END_IF

CASE _Step OF
	E_Ch1Ep1PrepareWaferTransferStep.MoveLiftPinAxis:
		IF NOT _CommandSubmitted THEN
			SubmitResult := M_StartDependency(
				ServiceId := E_Chamber1ServiceId.LiftPinAxisMoveAbs,
				Parameters := _LiftPinMoveParam);

			IF SubmitResult = E_ServiceCallSubmitResult.Queued THEN
				_CommandSubmitted := TRUE;
			ELSIF SubmitResult <> E_ServiceCallSubmitResult.Busy THEN
				M_FailSequence(
					ErrorCode := E_CompositeServiceErrorCode.InternalCallSubmitFailed,
					FailedServiceId := E_Chamber1ServiceId.LiftPinAxisMoveAbs,
					SourceErrorId := TO_UDINT(SubmitResult),
					Message := 'LiftPinAxis MoveAbs Start could not be queued.');
			END_IF
			RETURN;
		END_IF

		CommandState := M_GetDependencyCommandState(
			ServiceId := E_Chamber1ServiceId.LiftPinAxisMoveAbs);
		IF CommandState = E_ServiceInternalCommandState.Rejected THEN
			M_FailSequence(
				ErrorCode := E_CompositeServiceErrorCode.InternalCommandRejected,
				FailedServiceId := E_Chamber1ServiceId.LiftPinAxisMoveAbs,
				SourceErrorId := TO_UDINT(E_PackMLCommand.Start),
				Message := 'LiftPinAxis MoveAbs Start was rejected.');
		ELSIF (CommandState = E_ServiceInternalCommandState.Cancelled)
			OR (CommandState = E_ServiceInternalCommandState.None) THEN
			M_FailSequence(
				ErrorCode := E_CompositeServiceErrorCode.InvalidSequenceState,
				FailedServiceId := E_Chamber1ServiceId.LiftPinAxisMoveAbs,
				SourceErrorId := TO_UDINT(CommandState),
				Message := 'LiftPinAxis MoveAbs command state was lost.');
		ELSIF (CommandState = E_ServiceInternalCommandState.Accepted)
			AND M_GetDependencyServiceSnapshot(
				ServiceId := E_Chamber1ServiceId.LiftPinAxisMoveAbs,
				Snapshot => Snapshot)
			AND (Snapshot.PackMLOut.eStateCurrent = E_PackMLState.Complete) THEN
			_Step := E_Ch1Ep1PrepareWaferTransferStep.VacuumOff;
			_CommandSubmitted := FALSE;
		END_IF

	E_Ch1Ep1PrepareWaferTransferStep.VacuumOff:
		IF NOT _CommandSubmitted THEN
			SubmitResult := M_StartDependency(
				ServiceId := E_Chamber1ServiceId.VacuumOff,
				Parameters := _VacuumOffParam);

			IF SubmitResult = E_ServiceCallSubmitResult.Queued THEN
				_CommandSubmitted := TRUE;
			ELSIF SubmitResult <> E_ServiceCallSubmitResult.Busy THEN
				M_FailSequence(
					ErrorCode := E_CompositeServiceErrorCode.InternalCallSubmitFailed,
					FailedServiceId := E_Chamber1ServiceId.VacuumOff,
					SourceErrorId := TO_UDINT(SubmitResult),
					Message := 'VacuumOff Start could not be queued.');
			END_IF
			RETURN;
		END_IF

		CommandState := M_GetDependencyCommandState(
			ServiceId := E_Chamber1ServiceId.VacuumOff);
		IF CommandState = E_ServiceInternalCommandState.Rejected THEN
			M_FailSequence(
				ErrorCode := E_CompositeServiceErrorCode.InternalCommandRejected,
				FailedServiceId := E_Chamber1ServiceId.VacuumOff,
				SourceErrorId := TO_UDINT(E_PackMLCommand.Start),
				Message := 'VacuumOff Start was rejected.');
		ELSIF (CommandState = E_ServiceInternalCommandState.Cancelled)
			OR (CommandState = E_ServiceInternalCommandState.None) THEN
			M_FailSequence(
				ErrorCode := E_CompositeServiceErrorCode.InvalidSequenceState,
				FailedServiceId := E_Chamber1ServiceId.VacuumOff,
				SourceErrorId := TO_UDINT(CommandState),
				Message := 'VacuumOff command state was lost.');
		ELSIF (CommandState = E_ServiceInternalCommandState.Accepted)
			AND M_GetDependencyServiceSnapshot(
				ServiceId := E_Chamber1ServiceId.VacuumOff,
				Snapshot => Snapshot)
			AND (Snapshot.PackMLOut.eStateCurrent = E_PackMLState.Complete) THEN
			_Step := E_Ch1Ep1PrepareWaferTransferStep.Finish;
			_CommandSubmitted := FALSE;
		END_IF

	E_Ch1Ep1PrepareWaferTransferStep.Finish:
		H_OnCompositeExecute := E_PackMLHookResult.Done;

	ELSE
		M_FailSequence(
			ErrorCode := E_CompositeServiceErrorCode.InvalidSequenceState,
			FailedServiceId := ServiceId,
			SourceErrorId := TO_UDINT(_Step),
			Message := 'Endpoint1PrepareSendWafer entered an invalid sequence step.');
END_CASE
END_METHOD

END_FUNCTION_BLOCK

// ---- POUs/10_Chamber1/Services/FB_Chamber1PreparePositionService.TcPOU
FUNCTION_BLOCK FB_Chamber1PreparePositionService EXTENDS FB_CompositeServiceBase
VAR_INPUT
	Param : ST_Chamber1PreparePositionParam;
END_VAR
VAR
	_Step : E_Chamber1PreparePositionStep;
	_CommandSubmitted : BOOL;
	
	_LiftReadyParam : ST_Chamber1LiftPinAxisMoveAbsParam;
	_SpinAlignParam : ST_Chamber1SpinAxisMoveAbsParam;
	_LiftWorkParam : ST_Chamber1LiftPinAxisMoveAbsParam;
END_VAR

M_UpdateCompositeService();

METHOD PROTECTED H_DeclareServices
M_AddDependency(ServiceId := E_Chamber1ServiceId.LiftPinAxisMoveAbs);
M_AddDependency(ServiceId := E_Chamber1ServiceId.SpinAxisMoveAbs);
END_METHOD

METHOD PROTECTED H_GetExecuteSubState : UDINT
H_GetExecuteSubState := TO_UDINT(_Step);
END_METHOD

METHOD PROTECTED H_GetExecuteSubStateName : STRING(80)
H_GetExecuteSubStateName := TO_STRING(_Step);
END_METHOD

METHOD PROTECTED H_OnCompositeExecute : E_PackMLHookResult
VAR_INPUT
	bFirstScan : BOOL;
END_VAR
VAR
	SubmitResult : E_ServiceCallSubmitResult;
	CommandState : E_ServiceInternalCommandState;
	Snapshot : ST_ServiceExecutionSnapshot;

END_VAR
H_OnCompositeExecute := E_PackMLHookResult.Busy;

IF bFirstScan THEN
	_Step := E_Chamber1PreparePositionStep.LiftReady;
	_CommandSubmitted := FALSE;
END_IF

CASE _Step OF
	E_Chamber1PreparePositionStep.LiftReady:
	
		// Set command if not submitted
		IF NOT _CommandSubmitted THEN
			_LiftReadyParam.Position := Param.LiftReadyPosition;
			_LiftReadyParam.Velocity := Param.LiftReadyVelocity;
			_LiftReadyParam.Acceleration := Param.LiftReadyAcceleration;
			_LiftReadyParam.Deceleration := Param.LiftReadyDeceleration;

			SubmitResult := M_StartDependency(
				ServiceId := E_Chamber1ServiceId.LiftPinAxisMoveAbs,
				Parameters := _LiftReadyParam);
			
			// Submit successfully
			IF SubmitResult = E_ServiceCallSubmitResult.Queued THEN
				_CommandSubmitted := TRUE;
			
			// Submit failed
			ELSIF SubmitResult <> E_ServiceCallSubmitResult.Busy THEN
				M_FailSequence(ErrorCode := E_CompositeServiceErrorCode.InternalCallSubmitFailed,
					FailedServiceId := E_Chamber1ServiceId.LiftPinAxisMoveAbs,
					SourceErrorId := TO_UDINT(SubmitResult), Message := 'LiftReady Start could not be queued.');
			END_IF
			RETURN;
		END_IF
		
		// Check command result
		CommandState := M_GetDependencyCommandState(ServiceId := E_Chamber1ServiceId.LiftPinAxisMoveAbs);
		IF CommandState = E_ServiceInternalCommandState.Rejected THEN
			M_FailSequence(ErrorCode := E_CompositeServiceErrorCode.InternalCommandRejected,
				FailedServiceId := E_Chamber1ServiceId.LiftPinAxisMoveAbs,
				SourceErrorId := TO_UDINT(E_PackMLCommand.Start), Message := 'LiftReady Start was rejected.');
				
		ELSIF (CommandState = E_ServiceInternalCommandState.Cancelled)
			OR (CommandState = E_ServiceInternalCommandState.None) THEN
			M_FailSequence(ErrorCode := E_CompositeServiceErrorCode.InvalidSequenceState,
				FailedServiceId := E_Chamber1ServiceId.LiftPinAxisMoveAbs,
				SourceErrorId := TO_UDINT(CommandState), Message := 'LiftReady command state was lost.');
				
		ELSIF (CommandState = E_ServiceInternalCommandState.Accepted)
			AND M_GetDependencyServiceSnapshot(
				ServiceId := E_Chamber1ServiceId.LiftPinAxisMoveAbs, Snapshot => Snapshot)
			AND (Snapshot.PackMLOut.eStateCurrent = E_PackMLState.Complete) THEN
			
			// Transition
			_Step := E_Chamber1PreparePositionStep.SpinAlign;
			_CommandSubmitted := FALSE;
		END_IF

	E_Chamber1PreparePositionStep.SpinAlign:
	
		// Set command if not submitted
		IF NOT _CommandSubmitted THEN
			_SpinAlignParam.Position := Param.SpinAlignPosition;
			_SpinAlignParam.Velocity := Param.SpinAlignVelocity;
			_SpinAlignParam.Acceleration := Param.SpinAlignAcceleration;
			_SpinAlignParam.Deceleration := Param.SpinAlignDeceleration;

			SubmitResult := M_StartDependency(
				ServiceId := E_Chamber1ServiceId.SpinAxisMoveAbs,
				Parameters := _SpinAlignParam);
				
			IF SubmitResult = E_ServiceCallSubmitResult.Queued THEN
				_CommandSubmitted := TRUE;
				
			ELSIF SubmitResult <> E_ServiceCallSubmitResult.Busy THEN
				M_FailSequence(ErrorCode := E_CompositeServiceErrorCode.InternalCallSubmitFailed,
					FailedServiceId := E_Chamber1ServiceId.SpinAxisMoveAbs,
					SourceErrorId := TO_UDINT(SubmitResult), Message := 'SpinAlign Start could not be queued.');
			END_IF
			RETURN;
		END_IF
		
		// Check command result
		CommandState := M_GetDependencyCommandState(ServiceId := E_Chamber1ServiceId.SpinAxisMoveAbs);
		IF CommandState = E_ServiceInternalCommandState.Rejected THEN
			M_FailSequence(ErrorCode := E_CompositeServiceErrorCode.InternalCommandRejected,
				FailedServiceId := E_Chamber1ServiceId.SpinAxisMoveAbs,
				SourceErrorId := TO_UDINT(E_PackMLCommand.Start), Message := 'SpinAlign Start was rejected.');
				
		ELSIF (CommandState = E_ServiceInternalCommandState.Cancelled)
			OR (CommandState = E_ServiceInternalCommandState.None) THEN
			M_FailSequence(ErrorCode := E_CompositeServiceErrorCode.InvalidSequenceState,
				FailedServiceId := E_Chamber1ServiceId.SpinAxisMoveAbs,
				SourceErrorId := TO_UDINT(CommandState), Message := 'SpinAlign command state was lost.');
				
		ELSIF (CommandState = E_ServiceInternalCommandState.Accepted)
			AND M_GetDependencyServiceSnapshot(
				ServiceId := E_Chamber1ServiceId.SpinAxisMoveAbs, Snapshot => Snapshot)
			AND (Snapshot.PackMLOut.eStateCurrent = E_PackMLState.Complete) THEN
			
			// Transition
			_Step := E_Chamber1PreparePositionStep.ResetLift;
			_CommandSubmitted := FALSE;
		END_IF

	E_Chamber1PreparePositionStep.ResetLift:
		IF NOT _CommandSubmitted THEN
			SubmitResult := M_CommandDependency(
				ServiceId := E_Chamber1ServiceId.LiftPinAxisMoveAbs,
				Command := E_PackMLCommand.Reset);
				
			IF SubmitResult = E_ServiceCallSubmitResult.Queued THEN
				_CommandSubmitted := TRUE;
				
			ELSIF SubmitResult <> E_ServiceCallSubmitResult.Busy THEN
				M_FailSequence(ErrorCode := E_CompositeServiceErrorCode.InternalCallSubmitFailed,
					FailedServiceId := E_Chamber1ServiceId.LiftPinAxisMoveAbs,
					SourceErrorId := TO_UDINT(SubmitResult), Message := 'Lift Reset could not be queued.');
			END_IF
			RETURN;
		END_IF
		CommandState := M_GetDependencyCommandState(ServiceId := E_Chamber1ServiceId.LiftPinAxisMoveAbs);
		IF CommandState = E_ServiceInternalCommandState.Rejected THEN
			M_FailSequence(ErrorCode := E_CompositeServiceErrorCode.InternalCommandRejected,
				FailedServiceId := E_Chamber1ServiceId.LiftPinAxisMoveAbs,
				SourceErrorId := TO_UDINT(E_PackMLCommand.Reset), Message := 'Lift Reset was rejected.');
				
		ELSIF (CommandState = E_ServiceInternalCommandState.Cancelled)
			OR (CommandState = E_ServiceInternalCommandState.None) THEN
			M_FailSequence(ErrorCode := E_CompositeServiceErrorCode.InvalidSequenceState,
				FailedServiceId := E_Chamber1ServiceId.LiftPinAxisMoveAbs,
				SourceErrorId := TO_UDINT(CommandState), Message := 'Lift Reset command state was lost.');
				
		ELSIF (CommandState = E_ServiceInternalCommandState.Accepted)
			AND M_GetDependencyServiceSnapshot(
				ServiceId := E_Chamber1ServiceId.LiftPinAxisMoveAbs, Snapshot => Snapshot)
			AND (Snapshot.PackMLOut.eStateCurrent = E_PackMLState.Idle) THEN
			_Step := E_Chamber1PreparePositionStep.LiftWork;
			_CommandSubmitted := FALSE;
		END_IF

	E_Chamber1PreparePositionStep.LiftWork:
		IF NOT _CommandSubmitted THEN
			_LiftWorkParam.Position := Param.LiftWorkPosition;
			_LiftWorkParam.Velocity := Param.LiftWorkVelocity;
			_LiftWorkParam.Acceleration := Param.LiftWorkAcceleration;
			_LiftWorkParam.Deceleration := Param.LiftWorkDeceleration;

			SubmitResult := M_StartDependency(
				ServiceId := E_Chamber1ServiceId.LiftPinAxisMoveAbs,
				Parameters := _LiftWorkParam);
				
			IF SubmitResult = E_ServiceCallSubmitResult.Queued THEN
				_CommandSubmitted := TRUE;
				
			ELSIF SubmitResult <> E_ServiceCallSubmitResult.Busy THEN
				M_FailSequence(ErrorCode := E_CompositeServiceErrorCode.InternalCallSubmitFailed,
					FailedServiceId := E_Chamber1ServiceId.LiftPinAxisMoveAbs,
					SourceErrorId := TO_UDINT(SubmitResult), Message := 'LiftWork Start could not be queued.');
			END_IF
			RETURN;
		END_IF
		
		CommandState := M_GetDependencyCommandState(ServiceId := E_Chamber1ServiceId.LiftPinAxisMoveAbs);
		IF CommandState = E_ServiceInternalCommandState.Rejected THEN
			M_FailSequence(ErrorCode := E_CompositeServiceErrorCode.InternalCommandRejected,
				FailedServiceId := E_Chamber1ServiceId.LiftPinAxisMoveAbs,
				SourceErrorId := TO_UDINT(E_PackMLCommand.Start), Message := 'LiftWork Start was rejected.');
				
		ELSIF (CommandState = E_ServiceInternalCommandState.Cancelled)
			OR (CommandState = E_ServiceInternalCommandState.None) THEN
			M_FailSequence(ErrorCode := E_CompositeServiceErrorCode.InvalidSequenceState,
				FailedServiceId := E_Chamber1ServiceId.LiftPinAxisMoveAbs,
				SourceErrorId := TO_UDINT(CommandState), Message := 'LiftWork command state was lost.');
				
		ELSIF (CommandState = E_ServiceInternalCommandState.Accepted)
			AND M_GetDependencyServiceSnapshot(
				ServiceId := E_Chamber1ServiceId.LiftPinAxisMoveAbs, Snapshot => Snapshot)
			AND (Snapshot.PackMLOut.eStateCurrent = E_PackMLState.Complete) THEN
			
			_Step := E_Chamber1PreparePositionStep.Finish;
			_CommandSubmitted := FALSE;
		END_IF

	E_Chamber1PreparePositionStep.Finish:
		H_OnCompositeExecute := E_PackMLHookResult.Done;

	ELSE
		M_FailSequence(ErrorCode := E_CompositeServiceErrorCode.InvalidSequenceState,
			FailedServiceId := ServiceId, SourceErrorId := TO_UDINT(_Step),
			Message := 'PreparePosition entered an invalid sequence step.');
END_CASE
END_METHOD

END_FUNCTION_BLOCK

// ---- POUs/FB_ConfigRoot.TcPOU
FUNCTION_BLOCK FB_ConfigRoot EXTENDS FB_ApplicationConfigRoot
VAR
	_Chamber1ModuleConfigurationAdapter : FB_Chamber1ModuleConfigurationAdapter;
END_VAR

METHOD PROTECTED H_RegisterBaseUnits
M_RegisterBaseUnit(BaseUnit := GVL_IO.NC_Axis1);
M_RegisterBaseUnit(BaseUnit := GVL_IO.NC_Axis2);
END_METHOD

METHOD PROTECTED H_RegisterIo
VAR
	nChannel : DINT;
END_VAR
FOR nChannel := LOWER_BOUND(GVL_IO.Term4_EL1889.Chl, 1)
	TO UPPER_BOUND(GVL_IO.Term4_EL1889.Chl, 1) DO
	IF NOT M_RegisterIoNode(
		Variable := GVL_IO.Term4_EL1889.Chl[nChannel],
		Access := E_VariableAccess.ReadOnly) THEN
		RETURN;
	END_IF
END_FOR

FOR nChannel := LOWER_BOUND(GVL_IO.Term2_EL3602.Chl, 1)
	TO UPPER_BOUND(GVL_IO.Term2_EL3602.Chl, 1) DO
	IF NOT M_RegisterIoNode(
		Variable := GVL_IO.Term2_EL3602.Chl[nChannel],
		Access := E_VariableAccess.ReadOnly) THEN
		RETURN;
	END_IF
END_FOR

FOR nChannel := LOWER_BOUND(GVL_IO.Term3_EL2809.Chl, 1)
	TO UPPER_BOUND(GVL_IO.Term3_EL2809.Chl, 1) DO
	IF NOT M_RegisterIoNode(
		Variable := GVL_IO.Term3_EL2809.Chl[nChannel],
		Access := E_VariableAccess.WriteOnly) THEN
		RETURN;
	END_IF
END_FOR

// Register share memory data
M_RegisterIoNode(
		Variable := GVL_ShareMemory.bChamber1_Endpoint1_DoorClosed,
		Access := E_VariableAccess.ReadWrite);
M_RegisterIoNode(
		Variable := GVL_ShareMemory.bChamber1_VacuumOn,
		Access := E_VariableAccess.ReadWrite);
M_RegisterIoNode(
		Variable := GVL_ShareMemory.bRobotIsInChamber1,
		Access := E_VariableAccess.ReadWrite);
END_METHOD

METHOD PROTECTED H_RegisterModuleTypes
M_RegisterModuleType(
	ModuleTypeName := 'Chamber1',
	Adapter := _Chamber1ModuleConfigurationAdapter);
END_METHOD

METHOD PROTECTED H_RunModules
VAR_INPUT
	VariableNodeReader : I_VariableNodeReader;
END_VAR
VAR_IN_OUT CONSTANT
	SystemContext : ST_SystemContext;
END_VAR
VAR
	nModule : UINT;
END_VAR
FOR nModule := 1 TO Param_Config.MaxModulePerType DO
	IF GVL_Module.Chamber1_Runtime[nModule].Enabled
		AND GVL_Module.Chamber1_Runtime[nModule].Valid THEN
		GVL_Module.Chamber1[nModule](
			HeartbeatIndex := GVL_Module.Chamber1_Control[nModule].HeartbeatIndex,
			ModuleCtrl := GVL_Module.Chamber1_Control[nModule].ModuleCtrl,
			ServiceCtrl := GVL_Module.Chamber1_Control[nModule].ServiceCtrl,
			ServiceParam := GVL_Module.Chamber1_Control[nModule].ServiceParam,
			SystemContext := SystemContext,
			RuntimeConfig := GVL_Module.Chamber1_Runtime[nModule],
			VariableNodeReader := VariableNodeReader,
			SpinAxis_BaseUnit := GVL_Module.Chamber1_SpinAxis[nModule],
			LiftPinAxis_BaseUnit := GVL_Module.Chamber1_LiftPinAxis[nModule],
			ModuleStatus => GVL_Module.Chamber1_Control[nModule].ModuleStatus,
			ServiceStatus => GVL_Module.Chamber1_Control[nModule].ServiceStatus,
			ModuleAlarmList => GVL_Module.Chamber1_Control[nModule].ModuleAlarmList,
			ModuleDataList => GVL_Module.Chamber1_Control[nModule].ModuleDataList,
			ModuleVariableList => GVL_Module.Chamber1_Control[nModule].ModuleVariableList);
	END_IF
END_FOR
END_METHOD

END_FUNCTION_BLOCK
